LIN {X 0.108,Y -513.249,Z 696.655,A 0.000,B 0.000,C 90.000,E1 333.896} C_DIS
LIN {X -0.045,Y -530.728,Z 696.649,A 0.000,B 0.000,C 90.000,E1 332.743} C_DIS
LIN {X 0.068,Y -536.802,Z 696.646,A 0.000,B 0.000,C 90.000,E1 332.308} C_DIS
LIN {X -0.021,Y -544.293,Z 696.643,A 0.000,B 0.000,C 90.000,E1 331.769} C_DIS
LIN {X 0.058,Y -551.459,Z 696.640,A 0.000,B 0.000,C 90.000,E1 331.179} C_DIS
LIN {X -0.040,Y -558.208,Z 696.637,A 0.000,B 0.000,C 90.000,E1 330.589} C_DIS
LIN {X 0.004,Y -562.208,Z 696.635,A 0.000,B 0.000,C 90.000,E1 330.205} C_DIS
LIN {X -0.100,Y -567.315,Z 696.632,A 0.000,B 0.000,C 90.000,E1 329.715} C_DIS
LIN {X 0.042,Y -574.841,Z 696.627,A 0.000,B 0.000,C 90.000,E1 328.918} C_DIS
LIN {X -0.001,Y -583.472,Z 696.622,A 0.000,B 0.000,C 90.000,E1 327.995} C_DIS
LIN {X 0.085,Y -588.408,Z 696.619,A 0.000,B 0.000,C 90.000,E1 327.454} C_DIS
LIN {X 0.306,Y -596.576,Z 696.614,A 0.000,B 0.000,C 90.000,E1 326.501} C_DIS
LIN {X -0.095,Y -603.275,Z 696.610,A 0.000,B 0.000,C 90.000,E1 325.754} C_DIS
LIN {X -0.164,Y -609.504,Z 696.605,A 0.000,B 0.000,C 90.000,E1 324.975} C_DIS
LIN {X -0.135,Y -614.465,Z 696.602,A 0.000,B 0.000,C 90.000,E1 324.322} C_DIS
LIN {X -0.109,Y -620.766,Z 696.597,A 0.000,B 0.000,C 90.000,E1 323.417} C_DIS
LIN {X 0.004,Y -625.954,Z 696.592,A 0.000,B 0.000,C 90.000,E1 322.637} C_DIS
LIN {X 0.012,Y -633.084,Z 696.586,A 0.000,B 0.000,C 90.000,E1 321.492} C_DIS
LIN {X 0.145,Y -637.620,Z 696.582,A 0.000,B 0.000,C 90.000,E1 320.723} C_DIS
LIN {X -0.076,Y -641.917,Z 696.578,A 0.000,B 0.000,C 90.000,E1 319.989} C_DIS
LIN {X 0.082,Y -648.096,Z 696.571,A 0.000,B 0.000,C 90.000,E1 318.852} C_DIS
LIN {X -0.152,Y -653.942,Z 696.565,A 0.000,B 0.000,C 90.000,E1 317.757} C_DIS
LIN {X 0.212,Y -657.573,Z 696.561,A 0.000,B 0.000,C 90.000,E1 316.986} C_DIS
LIN {X -0.327,Y -660.960,Z 696.557,A 0.000,B 0.000,C 90.000,E1 316.296} C_DIS
LIN {X -0.383,Y -664.239,Z 696.553,A 0.000,B 0.000,C 90.000,E1 315.567} C_DIS
LIN {X 0.064,Y -668.154,Z 696.548,A 0.000,B 0.000,C 90.000,E1 314.555} C_DIS
LIN {X 0.123,Y -672.812,Z 696.541,A 0.000,B 0.000,C 90.000,E1 313.338} C_DIS
LIN {X 0.209,Y -676.430,Z 696.536,A 0.000,B 0.000,C 90.000,E1 312.366} C_DIS
LIN {X -0.126,Y -679.960,Z 696.530,A 0.000,B 0.000,C 90.000,E1 311.434} C_DIS
LIN {X 0.093,Y -683.151,Z 696.525,A 0.000,B 0.000,C 90.000,E1 310.458} C_DIS
LIN {X -0.079,Y -686.060,Z 696.520,A 0.000,B 0.000,C 90.000,E1 309.519} C_DIS
LIN {X 0.020,Y -687.452,Z 696.517,A 0.000,B 0.000,C 90.000,E1 309.036} C_DIS
LIN {X 0.279,Y -689.267,Z 696.513,A 0.000,B 0.000,C 90.000,E1 308.302} C_DIS
LIN {X 0.187,Y -691.415,Z 696.508,A 0.000,B 0.000,C 90.000,E1 307.363} C_DIS
LIN {X 0.068,Y -692.857,Z 696.504,A 0.000,B 0.000,C 90.000,E1 306.664} C_DIS
LIN {X -0.332,Y -695.101,Z 696.497,A 0.000,B 0.000,C 90.000,E1 305.518} C_DIS
LIN {X 0.160,Y -696.257,Z 696.493,A 0.000,B 0.000,C 90.000,E1 304.771} C_DIS
LIN {X 0.036,Y -698.131,Z 696.485,A 0.000,B 0.000,C 90.000,E1 303.372} C_DIS
LIN {X 0.229,Y -699.119,Z 696.480,A 0.000,B 0.000,C 90.000,E1 302.418} C_DIS
LIN {X -0.243,Y -700.440,Z 696.472,A 0.000,B 0.000,C 90.000,E1 301.052} C_DIS
LIN {X -0.053,Y -701.022,Z 696.469,A 0.000,B 0.000,C 90.000,E1 300.335} C_DIS
LIN {X -0.253,Y -701.671,Z 696.461,A 0.000,B 0.000,C 90.000,E1 298.949} C_DIS
LIN {X 0.101,Y -702.488,Z 696.450,A 0.000,B 0.000,C 90.000,E1 297.052} C_DIS
LIN {X -0.098,Y -703.278,Z 696.443,A 0.000,B 0.000,C 90.000,E1 295.668} C_DIS
LIN {X -0.168,Y -703.320,Z 696.440,A 0.000,B 0.000,C 90.000,E1 295.207} C_DIS
LIN {X 0.113,Y -703.122,Z 696.439,A 0.000,B 0.000,C 90.000,E1 294.951} C_DIS
LIN {X -0.259,Y -702.120,Z 696.436,A 0.000,B 0.000,C 90.000,E1 294.515} C_DIS
LIN {X 0.018,Y -701.136,Z 696.435,A 0.000,B 0.000,C 90.000,E1 294.259} C_DIS
LIN {X 0.007,Y -699.413,Z 696.434,A 0.000,B 0.000,C 90.000,E1 294.027} C_DIS
LIN {X 0.276,Y -697.550,Z 696.432,A 0.000,B 0.000,C 90.000,E1 293.770} C_DIS
LIN {X -0.231,Y -696.472,Z 696.432,A 0.000,B 0.000,C 90.000,E1 293.695} C_DIS
LIN {X -0.101,Y -694.838,Z 696.431,A 0.000,B 0.000,C 90.000,E1 293.567} C_DIS
LIN {X 0.346,Y -688.862,Z 696.429,A 0.000,B 0.000,C 90.000,E1 293.259} C_DIS
LIN {X 0.117,Y -686.900,Z 696.429,A 0.000,B 0.000,C 90.000,E1 293.206} C_DIS
LIN {X 0.010,Y -684.820,Z 696.429,A 0.000,B 0.000,C 90.000,E1 293.153} C_DIS
LIN {X -0.122,Y -678.094,Z 696.428,A 0.000,B 0.000,C 90.000,E1 293.025} C_DIS
LIN {X -0.139,Y -661.568,Z 696.427,A 0.000,B 0.000,C 90.000,E1 292.823} C_DIS
LIN {X 0.114,Y -647.822,Z 696.426,A 0.000,B 0.000,C 90.000,E1 292.589} C_DIS
LIN {X 0.091,Y -638.127,Z 696.425,A 0.000,B 0.000,C 90.000,E1 292.408} C_DIS
LIN {X 0.149,Y -624.755,Z 696.423,A 0.000,B 0.000,C 90.000,E1 292.099} C_DIS
LIN {X -0.052,Y -607.642,Z 696.420,A 0.000,B 0.000,C 90.000,E1 291.663} C_DIS
LIN {X -0.239,Y -576.587,Z 696.415,A 0.000,B 0.000,C 90.000,E1 290.737} C_DIS
LIN {X 0.266,Y -569.169,Z 696.414,A 0.000,B 0.000,C 90.000,E1 290.482} C_DIS
LIN {X 0.114,Y -563.221,Z 696.413,A 0.000,B 0.000,C 90.000,E1 290.301} C_DIS
LIN {X 0.212,Y -560.426,Z 696.412,A 0.000,B 0.000,C 90.000,E1 290.174} C_DIS
LIN {X 0.106,Y -558.042,Z 696.412,A 0.000,B 0.000,C 90.000,E1 290.066} C_DIS
LIN {X -0.099,Y -555.714,Z 696.410,A 0.000,B 0.000,C 90.000,E1 289.885} C_DIS
LIN {X -0.136,Y -555.678,Z 696.410,A 0.000,B 0.000,C 90.000,E1 289.885} C_DIS
LIN {X 0.246,Y -554.917,Z 696.409,A 0.000,B 0.000,C 90.000,E1 289.631} C_DIS
LIN {X 0.065,Y -554.334,Z 696.406,A 0.000,B 0.000,C 90.000,E1 289.087} C_DIS
LIN {X 0.062,Y -553.901,Z 696.398,A 0.000,B 0.000,C 90.000,E1 287.692} C_DIS
LIN {X -0.009,Y -553.252,Z 696.389,A 0.000,B 0.000,C 90.000,E1 286.024} C_DIS
LIN {X 0.070,Y -552.874,Z 696.383,A 0.000,B 0.000,C 90.000,E1 284.898} C_DIS
LIN {X -0.155,Y -552.256,Z 696.374,A 0.000,B 0.000,C 90.000,E1 283.244} C_DIS
LIN {X 0.018,Y -551.645,Z 696.366,A 0.000,B 0.000,C 90.000,E1 281.827} C_DIS
LIN {X 0.069,Y -550.859,Z 696.356,A 0.000,B 0.000,C 90.000,E1 280.141} C_DIS
LIN {X -0.298,Y -549.954,Z 696.344,A 0.000,B 0.000,C 90.000,E1 277.936} C_DIS
LIN {X -0.091,Y -549.215,Z 696.328,A 0.000,B 0.000,C 90.000,E1 275.106} C_DIS
LIN {X -0.203,Y -548.955,Z 696.317,A 0.000,B 0.000,C 90.000,E1 273.151} C_DIS
LIN {X -0.006,Y -548.668,Z 696.311,A 0.000,B 0.000,C 90.000,E1 272.007} C_DIS
LIN {X 0.160,Y -548.440,Z 696.307,A 0.000,B 0.000,C 90.000,E1 271.146} C_DIS
LIN {X -0.045,Y -547.378,Z 696.296,A 0.000,B 0.000,C 90.000,E1 269.198} C_DIS
LIN {X 0.235,Y -546.347,Z 696.286,A 0.000,B 0.000,C 90.000,E1 267.478} C_DIS
LIN {X -0.020,Y -545.246,Z 696.277,A 0.000,B 0.000,C 90.000,E1 265.812} C_DIS
LIN {X -0.227,Y -543.753,Z 696.266,A 0.000,B 0.000,C 90.000,E1 263.856} C_DIS
LIN {X -0.042,Y -542.813,Z 696.260,A 0.000,B 0.000,C 90.000,E1 262.704} C_DIS
LIN {X -0.193,Y -540.813,Z 696.248,A 0.000,B 0.000,C 90.000,E1 260.735} C_DIS
LIN {X -0.169,Y -538.511,Z 696.234,A 0.000,B 0.000,C 90.000,E1 258.173} C_DIS
LIN {X -0.123,Y -536.708,Z 696.223,A 0.000,B 0.000,C 90.000,E1 256.172} C_DIS
LIN {X 0.182,Y -536.028,Z 696.218,A 0.000,B 0.000,C 90.000,E1 255.283} C_DIS
LIN {X 0.249,Y -534.304,Z 696.209,A 0.000,B 0.000,C 90.000,E1 253.559} C_DIS
LIN {X -0.079,Y -532.474,Z 696.199,A 0.000,B 0.000,C 90.000,E1 251.873} C_DIS
LIN {X -0.152,Y -531.320,Z 696.193,A 0.000,B 0.000,C 90.000,E1 250.732} C_DIS
LIN {X -0.070,Y -530.084,Z 696.187,A 0.000,B 0.000,C 90.000,E1 249.571} C_DIS
LIN {X -0.133,Y -527.665,Z 696.177,A 0.000,B 0.000,C 90.000,E1 247.847} C_DIS
LIN {X 0.090,Y -525.999,Z 696.170,A 0.000,B 0.000,C 90.000,E1 246.666} C_DIS
LIN {X 0.119,Y -524.652,Z 696.166,A 0.000,B 0.000,C 90.000,E1 245.793} C_DIS
LIN {X -0.126,Y -521.764,Z 696.156,A 0.000,B 0.000,C 90.000,E1 244.076} C_DIS
LIN {X 0.218,Y -519.540,Z 696.149,A 0.000,B 0.000,C 90.000,E1 242.871} C_DIS
LIN {X -0.031,Y -516.692,Z 696.141,A 0.000,B 0.000,C 90.000,E1 241.435} C_DIS
LIN {X 0.016,Y -514.319,Z 696.135,A 0.000,B 0.000,C 90.000,E1 240.255} C_DIS
LIN {X -0.070,Y -511.228,Z 696.127,A 0.000,B 0.000,C 90.000,E1 238.791} C_DIS
LIN {X -0.219,Y -508.022,Z 696.118,A 0.000,B 0.000,C 90.000,E1 237.327} C_DIS
LIN {X 0.222,Y -505.390,Z 696.112,A 0.000,B 0.000,C 90.000,E1 236.087} C_DIS
LIN {X 0.096,Y -502.049,Z 696.104,A 0.000,B 0.000,C 90.000,E1 234.609} C_DIS
LIN {X 0.033,Y -499.257,Z 696.097,A 0.000,B 0.000,C 90.000,E1 233.417} C_DIS
LIN {X 0.223,Y -496.243,Z 696.090,A 0.000,B 0.000,C 90.000,E1 232.190} C_DIS
LIN {X 0.069,Y -490.251,Z 696.077,A 0.000,B 0.000,C 90.000,E1 229.784} C_DIS
LIN {X 0.022,Y -485.908,Z 696.066,A 0.000,B 0.000,C 90.000,E1 227.957} C_DIS
LIN {X -0.016,Y -481.004,Z 696.055,A 0.000,B 0.000,C 90.000,E1 225.810} C_DIS
LIN {X -0.189,Y -478.295,Z 696.048,A 0.000,B 0.000,C 90.000,E1 224.595} C_DIS
LIN {X 0.048,Y -474.759,Z 696.039,A 0.000,B 0.000,C 90.000,E1 223.014} C_DIS
LIN {X -0.103,Y -471.293,Z 696.030,A 0.000,B 0.000,C 90.000,E1 221.472} C_DIS
LIN {X 0.102,Y -467.176,Z 696.020,A 0.000,B 0.000,C 90.000,E1 219.564} C_DIS
LIN {X -0.020,Y -463.201,Z 696.009,A 0.000,B 0.000,C 90.000,E1 217.684} C_DIS
LIN {X -0.111,Y -458.072,Z 695.995,A 0.000,B 0.000,C 90.000,E1 215.152} C_DIS
LIN {X 0.306,Y -455.033,Z 695.986,A 0.000,B 0.000,C 90.000,E1 213.499} C_DIS
LIN {X 0.035,Y -451.969,Z 695.977,A 0.000,B 0.000,C 90.000,E1 211.926} C_DIS
LIN {X 0.012,Y -447.710,Z 695.965,A 0.000,B 0.000,C 90.000,E1 209.667} C_DIS
LIN {X 0.045,Y -443.555,Z 695.952,A 0.000,B 0.000,C 90.000,E1 207.385} C_DIS
LIN {X -0.122,Y -440.641,Z 695.943,A 0.000,B 0.000,C 90.000,E1 205.771} C_DIS
LIN {X -0.145,Y -437.670,Z 695.934,A 0.000,B 0.000,C 90.000,E1 204.131} C_DIS
LIN {X -0.168,Y -433.971,Z 695.923,A 0.000,B 0.000,C 90.000,E1 202.153} C_DIS
LIN {X -0.091,Y -430.969,Z 695.914,A 0.000,B 0.000,C 90.000,E1 200.482} C_DIS
LIN {X -0.028,Y -427.298,Z 695.903,A 0.000,B 0.000,C 90.000,E1 198.471} C_DIS
LIN {X -0.134,Y -423.137,Z 695.890,A 0.000,B 0.000,C 90.000,E1 196.134} C_DIS
LIN {X 0.011,Y -420.120,Z 695.880,A 0.000,B 0.000,C 90.000,E1 194.426} C_DIS
LIN {X -0.102,Y -415.938,Z 695.867,A 0.000,B 0.000,C 90.000,E1 192.063} C_DIS
LIN {X 0.217,Y -413.119,Z 695.857,A 0.000,B 0.000,C 90.000,E1 190.310} C_DIS
LIN {X 0.025,Y -409.762,Z 695.846,A 0.000,B 0.000,C 90.000,E1 188.276} C_DIS
LIN {X 0.049,Y -406.705,Z 695.835,A 0.000,B 0.000,C 90.000,E1 186.201} C_DIS
LIN {X -0.040,Y -403.260,Z 695.821,A 0.000,B 0.000,C 90.000,E1 183.784} C_DIS
LIN {X 0.025,Y -399.368,Z 695.804,A 0.000,B 0.000,C 90.000,E1 180.630} C_DIS
LIN {X -0.112,Y -395.946,Z 695.784,A 0.000,B 0.000,C 90.000,E1 177.135} C_DIS
LIN {X -0.171,Y -393.858,Z 695.768,A 0.000,B 0.000,C 90.000,E1 174.318} C_DIS
LIN {X 0.047,Y -392.119,Z 695.747,A 0.000,B 0.000,C 90.000,E1 170.387} C_DIS
LIN {X -0.203,Y -391.473,Z 695.733,A 0.000,B 0.000,C 90.000,E1 167.937} C_DIS
LIN {X 0.130,Y -390.914,Z 695.721,A 0.000,B 0.000,C 90.000,E1 165.755} C_DIS
LIN {X 0.146,Y -390.479,Z 695.705,A 0.000,B 0.000,C 90.000,E1 162.906} C_DIS
LIN {X -0.008,Y -390.447,Z 695.695,A 0.000,B 0.000,C 90.000,E1 161.148} C_DIS
LIN {X 0.061,Y -390.499,Z 695.681,A 0.000,B 0.000,C 90.000,E1 158.646} C_DIS
LIN {X -0.100,Y -390.667,Z 695.668,A 0.000,B 0.000,C 90.000,E1 156.177} C_DIS
LIN {X 0.213,Y -390.978,Z 695.654,A 0.000,B 0.000,C 90.000,E1 153.640} C_DIS
LIN {X 0.164,Y -391.240,Z 695.642,A 0.000,B 0.000,C 90.000,E1 151.513} C_DIS
LIN {X -0.185,Y -391.908,Z 695.628,A 0.000,B 0.000,C 90.000,E1 149.076} C_DIS
LIN {X 0.174,Y -392.559,Z 695.618,A 0.000,B 0.000,C 90.000,E1 147.248} C_DIS
LIN {X 0.153,Y -393.926,Z 695.604,A 0.000,B 0.000,C 90.000,E1 144.769} C_DIS
LIN {X 0.031,Y -394.813,Z 695.597,A 0.000,B 0.000,C 90.000,E1 143.371} C_DIS
LIN {X 0.035,Y -396.587,Z 695.585,A 0.000,B 0.000,C 90.000,E1 141.251} C_DIS
LIN {X 0.039,Y -398.612,Z 695.573,A 0.000,B 0.000,C 90.000,E1 139.138} C_DIS
LIN {X -0.021,Y -400.455,Z 695.563,A 0.000,B 0.000,C 90.000,E1 137.391} C_DIS
LIN {X -0.097,Y -401.201,Z 695.559,A 0.000,B 0.000,C 90.000,E1 136.701} C_DIS
LIN {X 0.108,Y -402.322,Z 695.556,A 0.000,B 0.000,C 90.000,E1 135.972} C_DIS
LIN {X -0.045,Y -404.292,Z 695.551,A 0.000,B 0.000,C 90.000,E1 135.121} C_DIS
LIN {X -0.117,Y -407.030,Z 695.547,A 0.000,B 0.000,C 90.000,E1 134.433} C_DIS
LIN {X 0.194,Y -409.182,Z 695.545,A 0.000,B 0.000,C 90.000,E1 134.028} C_DIS
LIN {X 0.022,Y -412.574,Z 695.542,A 0.000,B 0.000,C 90.000,E1 133.623} C_DIS
LIN {X -0.085,Y -418.142,Z 695.539,A 0.000,B 0.000,C 90.000,E1 133.056} C_DIS
LIN {X 0.040,Y -436.277,Z 695.530,A 0.000,B 0.000,C 90.000,E1 131.391} C_DIS
LIN {X -0.063,Y -454.811,Z 695.521,A 0.000,B 0.000,C 90.000,E1 129.850} C_DIS
LIN {X 0.035,Y -465.484,Z 695.516,A 0.000,B 0.000,C 90.000,E1 128.955} C_DIS
LIN {X 0.013,Y -474.374,Z 695.512,A 0.000,B 0.000,C 90.000,E1 128.177} C_DIS
LIN {X 0.078,Y -481.386,Z 695.509,A 0.000,B 0.000,C 90.000,E1 127.523} C_DIS
LIN {X -0.109,Y -488.508,Z 695.505,A 0.000,B 0.000,C 90.000,E1 126.870} C_DIS
LIN {X 0.152,Y -495.304,Z 695.501,A 0.000,B 0.000,C 90.000,E1 126.171} C_DIS
LIN {X 0.101,Y -502.112,Z 695.497,A 0.000,B 0.000,C 90.000,E1 125.471} C_DIS
LIN {X 0.044,Y -508.566,Z 695.493,A 0.000,B 0.000,C 90.000,E1 124.771} C_DIS
LIN {X 0.125,Y -513.389,Z 695.490,A 0.000,B 0.000,C 90.000,E1 124.199} C_DIS
LIN {X -0.011,Y -517.919,Z 695.487,A 0.000,B 0.000,C 90.000,E1 123.658} C_DIS
LIN {X 0.083,Y -522.141,Z 695.484,A 0.000,B 0.000,C 90.000,E1 123.086} C_DIS
LIN {X 0.009,Y -526.038,Z 695.481,A 0.000,B 0.000,C 90.000,E1 122.546} C_DIS
LIN {X -0.254,Y -530.643,Z 695.477,A 0.000,B 0.000,C 90.000,E1 121.878} C_DIS
LIN {X 0.146,Y -534.089,Z 695.474,A 0.000,B 0.000,C 90.000,E1 121.258} C_DIS
LIN {X 0.016,Y -538.708,Z 695.469,A 0.000,B 0.000,C 90.000,E1 120.413} C_DIS
LIN {X -0.128,Y -542.209,Z 695.465,A 0.000,B 0.000,C 90.000,E1 119.716} C_DIS
LIN {X -0.044,Y -545.486,Z 695.461,A 0.000,B 0.000,C 90.000,E1 118.999} C_DIS
LIN {X 0.071,Y -548.557,Z 695.457,A 0.000,B 0.000,C 90.000,E1 118.281} C_DIS
LIN {X -0.161,Y -551.986,Z 695.453,A 0.000,B 0.000,C 90.000,E1 117.462} C_DIS
LIN {X -0.102,Y -555.184,Z 695.448,A 0.000,B 0.000,C 90.000,E1 116.616} C_DIS
LIN {X 0.277,Y -559.133,Z 695.442,A 0.000,B 0.000,C 90.000,E1 115.463} C_DIS
LIN {X 0.164,Y -561.826,Z 695.437,A 0.000,B 0.000,C 90.000,E1 114.643} C_DIS
LIN {X 0.080,Y -564.293,Z 695.432,A 0.000,B 0.000,C 90.000,E1 113.823} C_DIS
LIN {X 0.128,Y -567.059,Z 695.426,A 0.000,B 0.000,C 90.000,E1 112.717} C_DIS
LIN {X -0.247,Y -568.297,Z 695.423,A 0.000,B 0.000,C 90.000,E1 112.206} C_DIS
LIN {X -0.139,Y -570.468,Z 695.417,A 0.000,B 0.000,C 90.000,E1 111.099} C_DIS
LIN {X 0.162,Y -572.974,Z 695.410,A 0.000,B 0.000,C 90.000,E1 109.704} C_DIS
LIN {X -0.032,Y -575.321,Z 695.402,A 0.000,B 0.000,C 90.000,E1 108.362} C_DIS
LIN {X 0.180,Y -577.652,Z 695.395,A 0.000,B 0.000,C 90.000,E1 106.985} C_DIS
LIN {X 0.222,Y -579.456,Z 695.388,A 0.000,B 0.000,C 90.000,E1 105.898} C_DIS
LIN {X -0.218,Y -581.581,Z 695.381,A 0.000,B 0.000,C 90.000,E1 104.592} C_DIS
LIN {X 0.173,Y -584.094,Z 695.372,A 0.000,B 0.000,C 90.000,E1 102.939} C_DIS
LIN {X -0.205,Y -586.524,Z 695.363,A 0.000,B 0.000,C 90.000,E1 101.366} C_DIS
LIN {X -0.096,Y -588.661,Z 695.356,A 0.000,B 0.000,C 90.000,E1 100.018} C_DIS
LIN {X 0.258,Y -590.190,Z 695.350,A 0.000,B 0.000,C 90.000,E1 98.916} C_DIS
LIN {X 0.049,Y -591.654,Z 695.344,A 0.000,B 0.000,C 90.000,E1 97.871} C_DIS
LIN {X 0.241,Y -593.679,Z 695.335,A 0.000,B 0.000,C 90.000,E1 96.258} C_DIS
LIN {X 0.213,Y -595.276,Z 695.328,A 0.000,B 0.000,C 90.000,E1 94.935} C_DIS
LIN {X 0.211,Y -596.785,Z 695.320,A 0.000,B 0.000,C 90.000,E1 93.612} C_DIS
LIN {X -0.036,Y -597.871,Z 695.314,A 0.000,B 0.000,C 90.000,E1 92.579} C_DIS
LIN {X -0.274,Y -598.771,Z 695.308,A 0.000,B 0.000,C 90.000,E1 91.547} C_DIS
LIN {X 0.083,Y -599.562,Z 695.303,A 0.000,B 0.000,C 90.000,E1 90.458} C_DIS
LIN {X 0.098,Y -600.276,Z 695.295,A 0.000,B 0.000,C 90.000,E1 89.141} C_DIS
LIN {X 0.138,Y -600.768,Z 695.288,A 0.000,B 0.000,C 90.000,E1 87.822} C_DIS
LIN {X -0.055,Y -601.030,Z 695.282,A 0.000,B 0.000,C 90.000,E1 86.788} C_DIS
LIN {X -0.003,Y -601.236,Z 695.275,A 0.000,B 0.000,C 90.000,E1 85.469} C_DIS
LIN {X -0.146,Y -601.240,Z 695.269,A 0.000,B 0.000,C 90.000,E1 84.432} C_DIS
LIN {X 0.315,Y -601.145,Z 695.263,A 0.000,B 0.000,C 90.000,E1 83.337} C_DIS
LIN {X 0.174,Y -600.969,Z 695.257,A 0.000,B 0.000,C 90.000,E1 82.299} C_DIS
LIN {X 0.111,Y -600.661,Z 695.252,A 0.000,B 0.000,C 90.000,E1 81.254} C_DIS
LIN {X 0.049,Y -600.044,Z 695.246,A 0.000,B 0.000,C 90.000,E1 80.208} C_DIS
LIN {X -0.023,Y -599.215,Z 695.240,A 0.000,B 0.000,C 90.000,E1 79.162} C_DIS
LIN {X 0.178,Y -598.089,Z 695.232,A 0.000,B 0.000,C 90.000,E1 77.825} C_DIS
LIN {X 0.185,Y -597.114,Z 695.227,A 0.000,B 0.000,C 90.000,E1 76.769} C_DIS
LIN {X -0.268,Y -595.454,Z 695.218,A 0.000,B 0.000,C 90.000,E1 75.227} C_DIS
LIN {X 0.123,Y -593.924,Z 695.211,A 0.000,B 0.000,C 90.000,E1 73.866} C_DIS
LIN {X 0.082,Y -592.318,Z 695.203,A 0.000,B 0.000,C 90.000,E1 72.543} C_DIS
LIN {X 0.013,Y -590.482,Z 695.196,A 0.000,B 0.000,C 90.000,E1 71.221} C_DIS
LIN {X -0.021,Y -588.015,Z 695.187,A 0.000,B 0.000,C 90.000,E1 69.625} C_DIS
LIN {X 0.156,Y -586.212,Z 695.181,A 0.000,B 0.000,C 90.000,E1 68.539} C_DIS
LIN {X -0.032,Y -584.174,Z 695.175,A 0.000,B 0.000,C 90.000,E1 67.486} C_DIS
LIN {X -0.015,Y -581.818,Z 695.169,A 0.000,B 0.000,C 90.000,E1 66.410} C_DIS
LIN {X -0.262,Y -579.215,Z 695.163,A 0.000,B 0.000,C 90.000,E1 65.357} C_DIS
LIN {X -0.161,Y -577.083,Z 695.159,A 0.000,B 0.000,C 90.000,E1 64.537} C_DIS
LIN {X -0.088,Y -574.755,Z 695.154,A 0.000,B 0.000,C 90.000,E1 63.717} C_DIS
LIN {X 0.216,Y -572.228,Z 695.149,A 0.000,B 0.000,C 90.000,E1 62.871} C_DIS
LIN {X 0.325,Y -568.637,Z 695.143,A 0.000,B 0.000,C 90.000,E1 61.769} C_DIS
LIN {X 0.069,Y -565.689,Z 695.139,A 0.000,B 0.000,C 90.000,E1 60.973} C_DIS
LIN {X 0.277,Y -562.505,Z 695.134,A 0.000,B 0.000,C 90.000,E1 60.127} C_DIS
LIN {X -0.037,Y -558.888,Z 695.130,A 0.000,B 0.000,C 90.000,E1 59.331} C_DIS
LIN {X 0.190,Y -555.551,Z 695.126,A 0.000,B 0.000,C 90.000,E1 58.614} C_DIS
LIN {X 0.027,Y -552.644,Z 695.123,A 0.000,B 0.000,C 90.000,E1 58.074} C_DIS
LIN {X 0.018,Y -548.514,Z 695.119,A 0.000,B 0.000,C 90.000,E1 57.375} C_DIS
LIN {X -0.321,Y -544.014,Z 695.115,A 0.000,B 0.000,C 90.000,E1 56.707} C_DIS
LIN {X 0.189,Y -540.056,Z 695.112,A 0.000,B 0.000,C 90.000,E1 56.087} C_DIS
LIN {X -0.082,Y -535.707,Z 695.109,A 0.000,B 0.000,C 90.000,E1 55.548} C_DIS
LIN {X 0.103,Y -532.117,Z 695.106,A 0.000,B 0.000,C 90.000,E1 55.102} C_DIS
LIN {X -0.213,Y -527.228,Z 695.103,A 0.000,B 0.000,C 90.000,E1 54.609} C_DIS
LIN {X 0.155,Y -522.068,Z 695.101,A 0.000,B 0.000,C 90.000,E1 54.069} C_DIS
LIN {X -0.166,Y -516.546,Z 695.098,A 0.000,B 0.000,C 90.000,E1 53.623} C_DIS
LIN {X 0.201,Y -511.623,Z 695.096,A 0.000,B 0.000,C 90.000,E1 53.210} C_DIS
LIN {X 0.236,Y -505.365,Z 695.093,A 0.000,B 0.000,C 90.000,E1 52.763} C_DIS
LIN {X -0.126,Y -498.968,Z 695.091,A 0.000,B 0.000,C 90.000,E1 52.396} C_DIS
LIN {X 0.068,Y -489.097,Z 695.088,A 0.000,B 0.000,C 90.000,E1 51.778} C_DIS
LIN {X -0.109,Y -474.324,Z 695.083,A 0.000,B 0.000,C 90.000,E1 50.964} C_DIS
LIN {X -0.007,Y -467.665,Z 695.081,A 0.000,B 0.000,C 90.000,E1 50.561} C_DIS
LIN {X -0.061,Y -457.921,Z 695.078,A 0.000,B 0.000,C 90.000,E1 49.989} C_DIS
LIN {X -0.011,Y -440.182,Z 695.072,A 0.000,B 0.000,C 90.000,E1 48.895} C_DIS
LIN {X 0.011,Y -431.973,Z 695.069,A 0.000,B 0.000,C 90.000,E1 48.366} C_DIS
LIN {X 0.061,Y -424.375,Z 695.066,A 0.000,B 0.000,C 90.000,E1 47.796} C_DIS
LIN {X 0.033,Y -424.361,Z 695.066,A 0.000,B 0.000,C 90.000,E1 47.796} C_DIS
LIN {X 0.137,Y -418.983,Z 695.050,A 0.000,B 0.000,C 90.000,E1 45.000} C_DIS
LIN {X 0.026,Y -418.304,Z 695.048,A 0.000,B 0.000,C 90.000,E1 44.676} C_DIS
LIN {X 0.079,Y -411.430,Z 695.031,A 0.000,B 0.000,C 90.000,E1 41.595} C_DIS
LIN {X -0.158,Y -411.330,Z 695.024,A 0.000,B 0.000,C 90.000,E1 40.253} C_DIS
LIN {X 0.019,Y -411.919,Z 695.004,A 0.000,B 0.000,C 90.000,E1 36.790} C_DIS
LIN {X -0.053,Y -412.776,Z 694.993,A 0.000,B 0.000,C 90.000,E1 34.739} C_DIS
LIN {X -0.001,Y -413.750,Z 694.982,A 0.000,B 0.000,C 90.000,E1 32.673} C_DIS
LIN {X 0.261,Y -414.647,Z 694.972,A 0.000,B 0.000,C 90.000,E1 30.924} C_DIS
LIN {X -0.235,Y -415.608,Z 694.963,A 0.000,B 0.000,C 90.000,E1 29.283} C_DIS
LIN {X -0.084,Y -417.030,Z 694.949,A 0.000,B 0.000,C 90.000,E1 26.873} C_DIS
LIN {X 0.104,Y -418.712,Z 694.936,A 0.000,B 0.000,C 90.000,E1 24.463} C_DIS
LIN {X 0.107,Y -421.365,Z 694.919,A 0.000,B 0.000,C 90.000,E1 21.408} C_DIS
LIN {X -0.199,Y -423.013,Z 694.910,A 0.000,B 0.000,C 90.000,E1 19.758} C_DIS
LIN {X -0.077,Y -424.691,Z 694.900,A 0.000,B 0.000,C 90.000,E1 18.055} C_DIS
LIN {X 0.013,Y -426.775,Z 694.889,A 0.000,B 0.000,C 90.000,E1 16.024} C_DIS
LIN {X 0.244,Y -429.414,Z 694.876,A 0.000,B 0.000,C 90.000,E1 13.647} C_DIS
LIN {X 0.027,Y -431.453,Z 694.867,A 0.000,B 0.000,C 90.000,E1 12.007} C_DIS
LIN {X 0.093,Y -434.331,Z 694.854,A 0.000,B 0.000,C 90.000,E1 9.670} C_DIS
LIN {X -0.125,Y -438.203,Z 694.837,A 0.000,B 0.000,C 90.000,E1 6.720} C_DIS
LIN {X -0.012,Y -441.878,Z 694.823,A 0.000,B 0.000,C 90.000,E1 4.073} C_DIS
LIN {X -0.127,Y -446.523,Z 694.806,A 0.000,B 0.000,C 90.000,E1 1.146} C_DIS
LIN {X 0.061,Y -451.737,Z 694.790,A 0.000,B 0.000,C 90.000,E1 358.165} C_DIS
LIN {X 0.181,Y -455.413,Z 694.779,A 0.000,B 0.000,C 90.000,E1 356.216} C_DIS
LIN {X -0.236,Y -458.539,Z 694.770,A 0.000,B 0.000,C 90.000,E1 354.666} C_DIS
LIN {X 0.177,Y -461.137,Z 694.763,A 0.000,B 0.000,C 90.000,E1 353.337} C_DIS
LIN {X 0.164,Y -464.841,Z 694.753,A 0.000,B 0.000,C 90.000,E1 351.432} C_DIS
LIN {X 0.104,Y -467.813,Z 694.744,A 0.000,B 0.000,C 90.000,E1 349.859} C_DIS
LIN {X 0.106,Y -470.644,Z 694.735,A 0.000,B 0.000,C 90.000,E1 348.285} C_DIS
LIN {X 0.255,Y -473.485,Z 694.726,A 0.000,B 0.000,C 90.000,E1 346.700} C_DIS
LIN {X -0.051,Y -476.955,Z 694.716,A 0.000,B 0.000,C 90.000,E1 344.866} C_DIS
LIN {X 0.150,Y -481.136,Z 694.704,A 0.000,B 0.000,C 90.000,E1 342.670} C_DIS
LIN {X -0.029,Y -484.162,Z 694.695,A 0.000,B 0.000,C 90.000,E1 341.148} C_DIS
LIN {X -0.140,Y -487.297,Z 694.687,A 0.000,B 0.000,C 90.000,E1 339.625} C_DIS
LIN {X -0.171,Y -491.077,Z 694.677,A 0.000,B 0.000,C 90.000,E1 337.794} C_DIS
LIN {X 0.164,Y -493.752,Z 694.670,A 0.000,B 0.000,C 90.000,E1 336.538} C_DIS
LIN {X 0.252,Y -495.390,Z 694.666,A 0.000,B 0.000,C 90.000,E1 335.921} C_DIS
LIN {X -0.090,Y -497.607,Z 694.663,A 0.000,B 0.000,C 90.000,E1 335.357} C_DIS
LIN {X 0.009,Y -499.063,Z 694.661,A 0.000,B 0.000,C 90.000,E1 335.049} C_DIS
LIN {X 0.055,Y -501.270,Z 694.660,A 0.000,B 0.000,C 90.000,E1 334.717} C_DIS
LIN {X 0.074,Y -505.386,Z 694.657,A 0.000,B 0.000,C 90.000,E1 334.280} C_DIS
LIN {X 0.145,Y -510.759,Z 694.655,A 0.000,B 0.000,C 90.000,E1 333.845} C_DIS
LIN {X 0.160,Y -517.047,Z 694.652,A 0.000,B 0.000,C 90.000,E1 333.384} C_DIS
LIN {X 0.019,Y -529.596,Z 694.648,A 0.000,B 0.000,C 90.000,E1 332.564} C_DIS
LIN {X 0.140,Y -537.285,Z 694.645,A 0.000,B 0.000,C 90.000,E1 332.025} C_DIS
LIN {X -0.213,Y -544.685,Z 694.642,A 0.000,B 0.000,C 90.000,E1 331.513} C_DIS
LIN {X -0.189,Y -550.344,Z 694.639,A 0.000,B 0.000,C 90.000,E1 331.051} C_DIS
LIN {X 0.119,Y -557.227,Z 694.636,A 0.000,B 0.000,C 90.000,E1 330.411} C_DIS
LIN {X -0.002,Y -563.949,Z 694.632,A 0.000,B 0.000,C 90.000,E1 329.793} C_DIS
LIN {X 0.083,Y -572.921,Z 694.627,A 0.000,B 0.000,C 90.000,E1 328.869} C_DIS
LIN {X 0.012,Y -581.672,Z 694.622,A 0.000,B 0.000,C 90.000,E1 327.946} C_DIS
LIN {X -0.115,Y -587.830,Z 694.618,A 0.000,B 0.000,C 90.000,E1 327.296} C_DIS
LIN {X 0.117,Y -596.054,Z 694.613,A 0.000,B 0.000,C 90.000,E1 326.342} C_DIS
LIN {X -0.063,Y -604.011,Z 694.608,A 0.000,B 0.000,C 90.000,E1 325.435} C_DIS
LIN {X -0.154,Y -611.229,Z 694.603,A 0.000,B 0.000,C 90.000,E1 324.529} C_DIS
LIN {X 0.064,Y -615.046,Z 694.600,A 0.000,B 0.000,C 90.000,E1 323.989} C_DIS
LIN {X 0.254,Y -620.453,Z 694.596,A 0.000,B 0.000,C 90.000,E1 323.210} C_DIS
LIN {X -0.110,Y -624.824,Z 694.592,A 0.000,B 0.000,C 90.000,E1 322.603} C_DIS
LIN {X 0.401,Y -631.292,Z 694.587,A 0.000,B 0.000,C 90.000,E1 321.537} C_DIS
LIN {X -0.252,Y -634.418,Z 694.584,A 0.000,B 0.000,C 90.000,E1 321.090} C_DIS
LIN {X -0.108,Y -639.621,Z 694.579,A 0.000,B 0.000,C 90.000,E1 320.194} C_DIS
LIN {X 0.020,Y -645.916,Z 694.573,A 0.000,B 0.000,C 90.000,E1 319.057} C_DIS
LIN {X -0.123,Y -649.291,Z 694.569,A 0.000,B 0.000,C 90.000,E1 318.447} C_DIS
LIN {X -0.294,Y -654.457,Z 694.564,A 0.000,B 0.000,C 90.000,E1 317.472} C_DIS
LIN {X 0.103,Y -656.901,Z 694.561,A 0.000,B 0.000,C 90.000,E1 316.944} C_DIS
LIN {X 0.009,Y -660.345,Z 694.557,A 0.000,B 0.000,C 90.000,E1 316.215} C_DIS
LIN {X -0.051,Y -663.645,Z 694.553,A 0.000,B 0.000,C 90.000,E1 315.486} C_DIS
LIN {X -0.078,Y -667.626,Z 694.547,A 0.000,B 0.000,C 90.000,E1 314.514} C_DIS
LIN {X -0.057,Y -671.427,Z 694.542,A 0.000,B 0.000,C 90.000,E1 313.542} C_DIS
LIN {X 0.068,Y -676.057,Z 694.535,A 0.000,B 0.000,C 90.000,E1 312.324} C_DIS
LIN {X -0.265,Y -679.597,Z 694.530,A 0.000,B 0.000,C 90.000,E1 311.391} C_DIS
LIN {X 0.359,Y -682.106,Z 694.526,A 0.000,B 0.000,C 90.000,E1 310.620} C_DIS
LIN {X -0.350,Y -685.122,Z 694.521,A 0.000,B 0.000,C 90.000,E1 309.725} C_DIS
LIN {X -0.111,Y -687.253,Z 694.517,A 0.000,B 0.000,C 90.000,E1 308.991} C_DIS
LIN {X 0.203,Y -689.622,Z 694.511,A 0.000,B 0.000,C 90.000,E1 308.016} C_DIS
LIN {X 0.064,Y -691.278,Z 694.507,A 0.000,B 0.000,C 90.000,E1 307.317} C_DIS
LIN {X 0.362,Y -692.734,Z 694.503,A 0.000,B 0.000,C 90.000,E1 306.583} C_DIS
LIN {X -0.042,Y -695.026,Z 694.497,A 0.000,B 0.000,C 90.000,E1 305.438} C_DIS
LIN {X -0.125,Y -696.218,Z 694.493,A 0.000,B 0.000,C 90.000,E1 304.739} C_DIS
LIN {X 0.319,Y -698.112,Z 694.485,A 0.000,B 0.000,C 90.000,E1 303.293} C_DIS
LIN {X -0.117,Y -698.897,Z 694.481,A 0.000,B 0.000,C 90.000,E1 302.625} C_DIS
LIN {X -0.330,Y -700.497,Z 694.472,A 0.000,B 0.000,C 90.000,E1 301.003} C_DIS
LIN {X 0.219,Y -701.054,Z 694.468,A 0.000,B 0.000,C 90.000,E1 300.256} C_DIS
LIN {X 0.014,Y -701.741,Z 694.460,A 0.000,B 0.000,C 90.000,E1 298.871} C_DIS
LIN {X 0.042,Y -702.598,Z 694.450,A 0.000,B 0.000,C 90.000,E1 297.001} C_DIS
LIN {X -0.125,Y -703.305,Z 694.444,A 0.000,B 0.000,C 90.000,E1 295.848} C_DIS
LIN {X 0.439,Y -703.430,Z 694.441,A 0.000,B 0.000,C 90.000,E1 295.335} C_DIS
LIN {X -0.214,Y -703.397,Z 694.440,A 0.000,B 0.000,C 90.000,E1 295.155} C_DIS
LIN {X 0.069,Y -703.044,Z 694.438,A 0.000,B 0.000,C 90.000,E1 294.899} C_DIS
LIN {X -0.300,Y -701.959,Z 694.436,A 0.000,B 0.000,C 90.000,E1 294.463} C_DIS
LIN {X -0.161,Y -701.477,Z 694.435,A 0.000,B 0.000,C 90.000,E1 294.335} C_DIS
LIN {X -0.023,Y -700.713,Z 694.435,A 0.000,B 0.000,C 90.000,E1 294.207} C_DIS
LIN {X -0.404,Y -696.897,Z 694.432,A 0.000,B 0.000,C 90.000,E1 293.770} C_DIS
LIN {X -0.273,Y -695.571,Z 694.431,A 0.000,B 0.000,C 90.000,E1 293.643} C_DIS
LIN {X -0.144,Y -693.432,Z 694.431,A 0.000,B 0.000,C 90.000,E1 293.515} C_DIS
LIN {X 0.053,Y -687.820,Z 694.429,A 0.000,B 0.000,C 90.000,E1 293.259} C_DIS
LIN {X -0.166,Y -685.468,Z 694.429,A 0.000,B 0.000,C 90.000,E1 293.206} C_DIS
LIN {X -0.322,Y -678.893,Z 694.428,A 0.000,B 0.000,C 90.000,E1 293.078} C_DIS
LIN {X 0.077,Y -661.290,Z 694.427,A 0.000,B 0.000,C 90.000,E1 292.823} C_DIS
LIN {X -0.284,Y -647.520,Z 694.426,A 0.000,B 0.000,C 90.000,E1 292.642} C_DIS
LIN {X -0.320,Y -637.894,Z 694.425,A 0.000,B 0.000,C 90.000,E1 292.461} C_DIS
LIN {X -0.294,Y -624.415,Z 694.423,A 0.000,B 0.000,C 90.000,E1 292.153} C_DIS
LIN {X 0.071,Y -607.299,Z 694.420,A 0.000,B 0.000,C 90.000,E1 291.663} C_DIS
LIN {X -0.186,Y -576.094,Z 694.415,A 0.000,B 0.000,C 90.000,E1 290.737} C_DIS
LIN {X 0.291,Y -568.636,Z 694.414,A 0.000,B 0.000,C 90.000,E1 290.482} C_DIS
LIN {X 0.125,Y -562.420,Z 694.413,A 0.000,B 0.000,C 90.000,E1 290.301} C_DIS
LIN {X -0.240,Y -557.929,Z 694.412,A 0.000,B 0.000,C 90.000,E1 290.120} C_DIS
LIN {X 0.110,Y -555.662,Z 694.411,A 0.000,B 0.000,C 90.000,E1 289.885} C_DIS
LIN {X 0.073,Y -555.636,Z 694.411,A 0.000,B 0.000,C 90.000,E1 289.885} C_DIS
LIN {X 0.271,Y -554.841,Z 694.409,A 0.000,B 0.000,C 90.000,E1 289.631} C_DIS
LIN {X -0.269,Y -554.389,Z 694.407,A 0.000,B 0.000,C 90.000,E1 289.268} C_DIS
LIN {X 0.256,Y -553.944,Z 694.399,A 0.000,B 0.000,C 90.000,E1 287.819} C_DIS
LIN {X -0.073,Y -553.195,Z 694.388,A 0.000,B 0.000,C 90.000,E1 285.898} C_DIS
LIN {X -0.116,Y -552.927,Z 694.384,A 0.000,B 0.000,C 90.000,E1 285.064} C_DIS
LIN {X 0.186,Y -552.293,Z 694.374,A 0.000,B 0.000,C 90.000,E1 283.355} C_DIS
LIN {X 0.239,Y -551.691,Z 694.367,A 0.000,B 0.000,C 90.000,E1 281.951} C_DIS
LIN {X -0.031,Y -550.765,Z 694.356,A 0.000,B 0.000,C 90.000,E1 280.018} C_DIS
LIN {X 0.131,Y -549.867,Z 694.343,A 0.000,B 0.000,C 90.000,E1 277.757} C_DIS
LIN {X 0.226,Y -549.232,Z 694.329,A 0.000,B 0.000,C 90.000,E1 275.220} C_DIS
LIN {X 0.081,Y -548.990,Z 694.318,A 0.000,B 0.000,C 90.000,E1 273.269} C_DIS
LIN {X -0.241,Y -548.751,Z 694.312,A 0.000,B 0.000,C 90.000,E1 272.178} C_DIS
LIN {X -0.023,Y -548.395,Z 694.306,A 0.000,B 0.000,C 90.000,E1 271.031} C_DIS
LIN {X 0.271,Y -547.488,Z 694.296,A 0.000,B 0.000,C 90.000,E1 269.312} C_DIS
LIN {X 0.010,Y -546.474,Z 694.287,A 0.000,B 0.000,C 90.000,E1 267.650} C_DIS
LIN {X -0.279,Y -545.392,Z 694.278,A 0.000,B 0.000,C 90.000,E1 265.988} C_DIS
LIN {X 0.002,Y -544.292,Z 694.270,A 0.000,B 0.000,C 90.000,E1 264.546} C_DIS
LIN {X 0.200,Y -543.482,Z 694.263,A 0.000,B 0.000,C 90.000,E1 263.394} C_DIS
LIN {X -0.159,Y -542.381,Z 694.257,A 0.000,B 0.000,C 90.000,E1 262.299} C_DIS
LIN {X 0.137,Y -540.662,Z 694.248,A 0.000,B 0.000,C 90.000,E1 260.566} C_DIS
LIN {X 0.254,Y -538.412,Z 694.234,A 0.000,B 0.000,C 90.000,E1 257.993} C_DIS
LIN {X 0.302,Y -536.615,Z 694.222,A 0.000,B 0.000,C 90.000,E1 255.992} C_DIS
LIN {X -0.049,Y -535.893,Z 694.218,A 0.000,B 0.000,C 90.000,E1 255.172} C_DIS
LIN {X -0.034,Y -534.476,Z 694.210,A 0.000,B 0.000,C 90.000,E1 253.740} C_DIS
LIN {X 0.148,Y -532.653,Z 694.200,A 0.000,B 0.000,C 90.000,E1 252.000} C_DIS
LIN {X 0.266,Y -531.195,Z 694.192,A 0.000,B 0.000,C 90.000,E1 250.550} C_DIS
LIN {X -0.151,Y -529.926,Z 694.186,A 0.000,B 0.000,C 90.000,E1 249.444} C_DIS
LIN {X -0.036,Y -527.113,Z 694.175,A 0.000,B 0.000,C 90.000,E1 247.411} C_DIS
LIN {X 0.179,Y -525.411,Z 694.168,A 0.000,B 0.000,C 90.000,E1 246.230} C_DIS
LIN {X -0.273,Y -522.510,Z 694.158,A 0.000,B 0.000,C 90.000,E1 244.537} C_DIS
LIN {X -0.064,Y -520.978,Z 694.154,A 0.000,B 0.000,C 90.000,E1 243.640} C_DIS
LIN {X 0.172,Y -518.145,Z 694.145,A 0.000,B 0.000,C 90.000,E1 242.153} C_DIS
LIN {X -0.100,Y -515.285,Z 694.137,A 0.000,B 0.000,C 90.000,E1 240.717} C_DIS
LIN {X 0.273,Y -512.170,Z 694.129,A 0.000,B 0.000,C 90.000,E1 239.203} C_DIS
LIN {X 0.138,Y -509.033,Z 694.121,A 0.000,B 0.000,C 90.000,E1 237.740} C_DIS
LIN {X -0.110,Y -506.401,Z 694.114,A 0.000,B 0.000,C 90.000,E1 236.580} C_DIS
LIN {X -0.221,Y -503.070,Z 694.106,A 0.000,B 0.000,C 90.000,E1 235.102} C_DIS
LIN {X -0.265,Y -500.283,Z 694.099,A 0.000,B 0.000,C 90.000,E1 233.909} C_DIS
LIN {X 0.070,Y -498.126,Z 694.094,A 0.000,B 0.000,C 90.000,E1 232.970} C_DIS
LIN {X -0.061,Y -495.077,Z 694.088,A 0.000,B 0.000,C 90.000,E1 231.778} C_DIS
LIN {X -0.315,Y -490.630,Z 694.078,A 0.000,B 0.000,C 90.000,E1 229.989} C_DIS
LIN {X 0.019,Y -486.287,Z 694.067,A 0.000,B 0.000,C 90.000,E1 228.119} C_DIS
LIN {X -0.146,Y -482.021,Z 694.057,A 0.000,B 0.000,C 90.000,E1 226.296} C_DIS
LIN {X -0.181,Y -478.626,Z 694.049,A 0.000,B 0.000,C 90.000,E1 224.757} C_DIS
LIN {X 0.063,Y -475.069,Z 694.040,A 0.000,B 0.000,C 90.000,E1 223.176} C_DIS
LIN {X 0.090,Y -470.203,Z 694.028,A 0.000,B 0.000,C 90.000,E1 220.987} C_DIS
LIN {X -0.039,Y -466.112,Z 694.017,A 0.000,B 0.000,C 90.000,E1 219.116} C_DIS
LIN {X 0.061,Y -462.803,Z 694.009,A 0.000,B 0.000,C 90.000,E1 217.523} C_DIS
LIN {X 0.061,Y -457.733,Z 693.994,A 0.000,B 0.000,C 90.000,E1 214.978} C_DIS
LIN {X -0.001,Y -455.338,Z 693.987,A 0.000,B 0.000,C 90.000,E1 213.706} C_DIS
LIN {X -0.172,Y -451.644,Z 693.977,A 0.000,B 0.000,C 90.000,E1 211.799} C_DIS
LIN {X -0.275,Y -447.987,Z 693.966,A 0.000,B 0.000,C 90.000,E1 209.873} C_DIS
LIN {X -0.020,Y -443.819,Z 693.953,A 0.000,B 0.000,C 90.000,E1 207.564} C_DIS
LIN {X 0.017,Y -440.908,Z 693.944,A 0.000,B 0.000,C 90.000,E1 205.924} C_DIS
LIN {X 0.029,Y -437.325,Z 693.933,A 0.000,B 0.000,C 90.000,E1 203.951} C_DIS
LIN {X -0.230,Y -434.259,Z 693.924,A 0.000,B 0.000,C 90.000,E1 202.333} C_DIS
LIN {X 0.071,Y -430.660,Z 693.913,A 0.000,B 0.000,C 90.000,E1 200.301} C_DIS
LIN {X -0.008,Y -426.949,Z 693.902,A 0.000,B 0.000,C 90.000,E1 198.308} C_DIS
LIN {X -0.108,Y -422.812,Z 693.889,A 0.000,B 0.000,C 90.000,E1 195.969} C_DIS
LIN {X 0.145,Y -419.825,Z 693.879,A 0.000,B 0.000,C 90.000,E1 194.245} C_DIS
LIN {X 0.017,Y -415.660,Z 693.866,A 0.000,B 0.000,C 90.000,E1 191.883} C_DIS
LIN {X -0.155,Y -412.855,Z 693.857,A 0.000,B 0.000,C 90.000,E1 190.197} C_DIS
LIN {X 0.061,Y -409.558,Z 693.845,A 0.000,B 0.000,C 90.000,E1 188.106} C_DIS
LIN {X 0.084,Y -406.485,Z 693.834,A 0.000,B 0.000,C 90.000,E1 186.030} C_DIS
LIN {X 0.030,Y -403.544,Z 693.822,A 0.000,B 0.000,C 90.000,E1 183.955} C_DIS
LIN {X 0.103,Y -399.632,Z 693.805,A 0.000,B 0.000,C 90.000,E1 180.802} C_DIS
LIN {X 0.038,Y -396.479,Z 693.787,A 0.000,B 0.000,C 90.000,E1 177.650} C_DIS
LIN {X -0.031,Y -394.315,Z 693.771,A 0.000,B 0.000,C 90.000,E1 174.837} C_DIS
LIN {X 0.102,Y -392.308,Z 693.748,A 0.000,B 0.000,C 90.000,E1 170.566} C_DIS
LIN {X -0.069,Y -391.672,Z 693.734,A 0.000,B 0.000,C 90.000,E1 168.105} C_DIS
LIN {X 0.145,Y -391.246,Z 693.724,A 0.000,B 0.000,C 90.000,E1 166.297} C_DIS
LIN {X -0.170,Y -390.713,Z 693.706,A 0.000,B 0.000,C 90.000,E1 163.142} C_DIS
LIN {X 0.098,Y -390.652,Z 693.694,A 0.000,B 0.000,C 90.000,E1 160.967} C_DIS
LIN {X -0.011,Y -390.721,Z 693.683,A 0.000,B 0.000,C 90.000,E1 158.847} C_DIS
LIN {X 0.077,Y -390.803,Z 693.675,A 0.000,B 0.000,C 90.000,E1 157.411} C_DIS
LIN {X 0.015,Y -390.939,Z 693.667,A 0.000,B 0.000,C 90.000,E1 155.997} C_DIS
LIN {X -0.216,Y -391.180,Z 693.655,A 0.000,B 0.000,C 90.000,E1 153.896} C_DIS
LIN {X -0.065,Y -391.524,Z 693.641,A 0.000,B 0.000,C 90.000,E1 151.385} C_DIS
LIN {X -0.117,Y -392.012,Z 693.631,A 0.000,B 0.000,C 90.000,E1 149.616} C_DIS
LIN {X 0.241,Y -392.636,Z 693.621,A 0.000,B 0.000,C 90.000,E1 147.788} C_DIS
LIN {X 0.021,Y -394.369,Z 693.602,A 0.000,B 0.000,C 90.000,E1 144.276} C_DIS
LIN {X 0.236,Y -395.699,Z 693.592,A 0.000,B 0.000,C 90.000,E1 142.477} C_DIS
LIN {X -0.084,Y -398.190,Z 693.576,A 0.000,B 0.000,C 90.000,E1 139.703} C_DIS
LIN {X 0.217,Y -400.285,Z 693.564,A 0.000,B 0.000,C 90.000,E1 137.553} C_DIS
LIN {X -0.043,Y -401.391,Z 693.559,A 0.000,B 0.000,C 90.000,E1 136.539} C_DIS
LIN {X 0.164,Y -402.391,Z 693.555,A 0.000,B 0.000,C 90.000,E1 135.810} C_DIS
LIN {X 0.011,Y -404.285,Z 693.550,A 0.000,B 0.000,C 90.000,E1 134.960} C_DIS
LIN {X -0.189,Y -406.254,Z 693.547,A 0.000,B 0.000,C 90.000,E1 134.433} C_DIS
LIN {X 0.086,Y -409.232,Z 693.544,A 0.000,B 0.000,C 90.000,E1 133.866} C_DIS
LIN {X 0.025,Y -413.525,Z 693.541,A 0.000,B 0.000,C 90.000,E1 133.338} C_DIS
LIN {X -0.036,Y -419.627,Z 693.537,A 0.000,B 0.000,C 90.000,E1 132.732} C_DIS
LIN {X 0.139,Y -436.120,Z 693.529,A 0.000,B 0.000,C 90.000,E1 131.229} C_DIS
LIN {X 0.015,Y -456.247,Z 693.520,A 0.000,B 0.000,C 90.000,E1 129.564} C_DIS
LIN {X -0.112,Y -463.966,Z 693.516,A 0.000,B 0.000,C 90.000,E1 128.955} C_DIS
LIN {X -0.017,Y -471.361,Z 693.513,A 0.000,B 0.000,C 90.000,E1 128.302} C_DIS
LIN {X 0.043,Y -479.955,Z 693.509,A 0.000,B 0.000,C 90.000,E1 127.523} C_DIS
LIN {X 0.081,Y -486.857,Z 693.505,A 0.000,B 0.000,C 90.000,E1 126.870} C_DIS
LIN {X -0.277,Y -495.276,Z 693.500,A 0.000,B 0.000,C 90.000,E1 126.091} C_DIS
LIN {X -0.126,Y -500.698,Z 693.497,A 0.000,B 0.000,C 90.000,E1 125.518} C_DIS
LIN {X 0.007,Y -503.326,Z 693.496,A 0.000,B 0.000,C 90.000,E1 125.231} C_DIS
LIN {X -0.235,Y -508.503,Z 693.493,A 0.000,B 0.000,C 90.000,E1 124.692} C_DIS
LIN {X 0.070,Y -513.546,Z 693.489,A 0.000,B 0.000,C 90.000,E1 124.072} C_DIS
LIN {X 0.093,Y -517.272,Z 693.487,A 0.000,B 0.000,C 90.000,E1 123.627} C_DIS
LIN {X -0.288,Y -522.653,Z 693.483,A 0.000,B 0.000,C 90.000,E1 122.959} C_DIS
LIN {X 0.190,Y -526.741,Z 693.480,A 0.000,B 0.000,C 90.000,E1 122.339} C_DIS
LIN {X -0.008,Y -529.756,Z 693.477,A 0.000,B 0.000,C 90.000,E1 121.926} C_DIS
LIN {X 0.085,Y -534.896,Z 693.473,A 0.000,B 0.000,C 90.000,E1 121.052} C_DIS
LIN {X -0.352,Y -537.329,Z 693.470,A 0.000,B 0.000,C 90.000,E1 120.669} C_DIS
LIN {X -0.062,Y -541.622,Z 693.466,A 0.000,B 0.000,C 90.000,E1 119.795} C_DIS
LIN {X 0.020,Y -544.973,Z 693.462,A 0.000,B 0.000,C 90.000,E1 119.077} C_DIS
LIN {X 0.133,Y -548.118,Z 693.458,A 0.000,B 0.000,C 90.000,E1 118.359} C_DIS
LIN {X -0.080,Y -552.718,Z 693.451,A 0.000,B 0.000,C 90.000,E1 117.257} C_DIS
LIN {X -0.016,Y -555.895,Z 693.447,A 0.000,B 0.000,C 90.000,E1 116.411} C_DIS
LIN {X -0.166,Y -558.894,Z 693.442,A 0.000,B 0.000,C 90.000,E1 115.591} C_DIS
LIN {X -0.283,Y -561.655,Z 693.438,A 0.000,B 0.000,C 90.000,E1 114.771} C_DIS
LIN {X -0.051,Y -564.953,Z 693.431,A 0.000,B 0.000,C 90.000,E1 113.643} C_DIS
LIN {X -0.106,Y -567.042,Z 693.427,A 0.000,B 0.000,C 90.000,E1 112.823} C_DIS
LIN {X -0.174,Y -568.327,Z 693.424,A 0.000,B 0.000,C 90.000,E1 112.280} C_DIS
LIN {X -0.242,Y -571.088,Z 693.416,A 0.000,B 0.000,C 90.000,E1 110.918} C_DIS
LIN {X -0.094,Y -573.085,Z 693.410,A 0.000,B 0.000,C 90.000,E1 109.812} C_DIS
LIN {X 0.251,Y -575.458,Z 693.403,A 0.000,B 0.000,C 90.000,E1 108.417} C_DIS
LIN {X -0.091,Y -577.822,Z 693.395,A 0.000,B 0.000,C 90.000,E1 107.094} C_DIS
LIN {X 0.159,Y -580.080,Z 693.387,A 0.000,B 0.000,C 90.000,E1 105.717} C_DIS
LIN {X -0.082,Y -581.834,Z 693.381,A 0.000,B 0.000,C 90.000,E1 104.662} C_DIS
LIN {X -0.243,Y -584.350,Z 693.372,A 0.000,B 0.000,C 90.000,E1 103.063} C_DIS
LIN {X -0.241,Y -587.280,Z 693.362,A 0.000,B 0.000,C 90.000,E1 101.186} C_DIS
LIN {X -0.227,Y -589.417,Z 693.355,A 0.000,B 0.000,C 90.000,E1 99.849} C_DIS
LIN {X -0.177,Y -591.319,Z 693.347,A 0.000,B 0.000,C 90.000,E1 98.511} C_DIS
LIN {X -0.183,Y -593.099,Z 693.340,A 0.000,B 0.000,C 90.000,E1 97.182} C_DIS
LIN {X -0.161,Y -594.778,Z 693.332,A 0.000,B 0.000,C 90.000,E1 95.853} C_DIS
LIN {X 0.045,Y -596.704,Z 693.324,A 0.000,B 0.000,C 90.000,E1 94.245} C_DIS
LIN {X 0.062,Y -598.148,Z 693.316,A 0.000,B 0.000,C 90.000,E1 92.922} C_DIS
LIN {X -0.193,Y -599.141,Z 693.310,A 0.000,B 0.000,C 90.000,E1 91.892} C_DIS
LIN {X -0.172,Y -600.116,Z 693.303,A 0.000,B 0.000,C 90.000,E1 90.573} C_DIS
LIN {X -0.147,Y -600.835,Z 693.296,A 0.000,B 0.000,C 90.000,E1 89.255} C_DIS
LIN {X -0.097,Y -601.367,Z 693.289,A 0.000,B 0.000,C 90.000,E1 87.936} C_DIS
LIN {X -0.313,Y -601.627,Z 693.283,A 0.000,B 0.000,C 90.000,E1 86.906} C_DIS
LIN {X -0.217,Y -601.823,Z 693.275,A 0.000,B 0.000,C 90.000,E1 85.584} C_DIS
LIN {X 0.249,Y -601.835,Z 693.270,A 0.000,B 0.000,C 90.000,E1 84.489} C_DIS
LIN {X 0.122,Y -601.746,Z 693.264,A 0.000,B 0.000,C 90.000,E1 83.451} C_DIS
LIN {X 0.214,Y -601.459,Z 693.256,A 0.000,B 0.000,C 90.000,E1 82.129} C_DIS
LIN {X 0.154,Y -601.106,Z 693.251,A 0.000,B 0.000,C 90.000,E1 81.084} C_DIS
LIN {X 0.094,Y -600.457,Z 693.245,A 0.000,B 0.000,C 90.000,E1 80.038} C_DIS
LIN {X -0.253,Y -598.911,Z 693.234,A 0.000,B 0.000,C 90.000,E1 78.229} C_DIS
LIN {X 0.066,Y -597.638,Z 693.227,A 0.000,B 0.000,C 90.000,E1 76.881} C_DIS
LIN {X -0.078,Y -596.222,Z 693.220,A 0.000,B 0.000,C 90.000,E1 75.574} C_DIS
LIN {X -0.099,Y -595.067,Z 693.214,A 0.000,B 0.000,C 90.000,E1 74.519} C_DIS
LIN {X 0.143,Y -593.085,Z 693.205,A 0.000,B 0.000,C 90.000,E1 72.906} C_DIS
LIN {X -0.162,Y -591.682,Z 693.199,A 0.000,B 0.000,C 90.000,E1 71.873} C_DIS
LIN {X -0.239,Y -589.706,Z 693.192,A 0.000,B 0.000,C 90.000,E1 70.550} C_DIS
LIN {X -0.161,Y -587.540,Z 693.184,A 0.000,B 0.000,C 90.000,E1 69.209} C_DIS
LIN {X 0.089,Y -585.075,Z 693.177,A 0.000,B 0.000,C 90.000,E1 67.847} C_DIS
LIN {X 0.022,Y -583.397,Z 693.173,A 0.000,B 0.000,C 90.000,E1 67.050} C_DIS
LIN {X 0.029,Y -580.805,Z 693.167,A 0.000,B 0.000,C 90.000,E1 65.973} C_DIS
LIN {X 0.046,Y -579.512,Z 693.164,A 0.000,B 0.000,C 90.000,E1 65.433} C_DIS
LIN {X 0.144,Y -577.356,Z 693.159,A 0.000,B 0.000,C 90.000,E1 64.613} C_DIS
LIN {X -0.046,Y -575.005,Z 693.155,A 0.000,B 0.000,C 90.000,E1 63.819} C_DIS
LIN {X 0.006,Y -572.442,Z 693.150,A 0.000,B 0.000,C 90.000,E1 62.999} C_DIS
LIN {X 0.120,Y -568.807,Z 693.144,A 0.000,B 0.000,C 90.000,E1 61.897} C_DIS
LIN {X -0.132,Y -565.838,Z 693.139,A 0.000,B 0.000,C 90.000,E1 61.101} C_DIS
LIN {X 0.080,Y -562.646,Z 693.135,A 0.000,B 0.000,C 90.000,E1 60.255} C_DIS
LIN {X 0.250,Y -559.018,Z 693.130,A 0.000,B 0.000,C 90.000,E1 59.410} C_DIS
LIN {X 0.002,Y -555.658,Z 693.126,A 0.000,B 0.000,C 90.000,E1 58.742} C_DIS
LIN {X 0.018,Y -551.917,Z 693.122,A 0.000,B 0.000,C 90.000,E1 58.043} C_DIS
LIN {X 0.173,Y -547.616,Z 693.119,A 0.000,B 0.000,C 90.000,E1 57.327} C_DIS
LIN {X -0.045,Y -543.982,Z 693.115,A 0.000,B 0.000,C 90.000,E1 56.786} C_DIS
LIN {X 0.012,Y -540.021,Z 693.112,A 0.000,B 0.000,C 90.000,E1 56.215} C_DIS
LIN {X -0.256,Y -535.585,Z 693.109,A 0.000,B 0.000,C 90.000,E1 55.674} C_DIS
LIN {X 0.056,Y -529.628,Z 693.106,A 0.000,B 0.000,C 90.000,E1 54.975} C_DIS
LIN {X 0.135,Y -525.717,Z 693.103,A 0.000,B 0.000,C 90.000,E1 54.562} C_DIS
LIN {X 0.049,Y -521.667,Z 693.101,A 0.000,B 0.000,C 90.000,E1 54.196} C_DIS
LIN {X 0.300,Y -516.226,Z 693.099,A 0.000,B 0.000,C 90.000,E1 53.703} C_DIS
LIN {X 0.243,Y -511.263,Z 693.096,A 0.000,B 0.000,C 90.000,E1 53.336} C_DIS
LIN {X 0.058,Y -503.728,Z 693.094,A 0.000,B 0.000,C 90.000,E1 52.844} C_DIS
LIN {X 0.078,Y -497.178,Z 693.091,A 0.000,B 0.000,C 90.000,E1 52.431} C_DIS
LIN {X 0.300,Y -487.334,Z 693.088,A 0.000,B 0.000,C 90.000,E1 51.823} C_DIS
LIN {X 0.156,Y -474.003,Z 693.084,A 0.000,B 0.000,C 90.000,E1 51.090} C_DIS
LIN {X 0.097,Y -462.819,Z 693.080,A 0.000,B 0.000,C 90.000,E1 50.436} C_DIS
LIN {X 0.186,Y -438.355,Z 693.072,A 0.000,B 0.000,C 90.000,E1 48.933} C_DIS
LIN {X 0.072,Y -431.860,Z 693.070,A 0.000,B 0.000,C 90.000,E1 48.528} C_DIS
LIN {X 0.202,Y -424.877,Z 693.067,A 0.000,B 0.000,C 90.000,E1 48.000} C_DIS
LIN {X 0.174,Y -424.843,Z 693.067,A 0.000,B 0.000,C 90.000,E1 48.000} C_DIS
LIN {X 0.028,Y -418.678,Z 693.049,A 0.000,B 0.000,C 90.000,E1 44.838} C_DIS
LIN {X 0.096,Y -411.760,Z 693.032,A 0.000,B 0.000,C 90.000,E1 41.757} C_DIS
LIN {X 0.063,Y -411.892,Z 693.015,A 0.000,B 0.000,C 90.000,E1 38.669} C_DIS
LIN {X 0.082,Y -413.011,Z 692.996,A 0.000,B 0.000,C 90.000,E1 35.231} C_DIS
LIN {X 0.144,Y -413.970,Z 692.984,A 0.000,B 0.000,C 90.000,E1 33.166} C_DIS
LIN {X 0.005,Y -415.062,Z 692.973,A 0.000,B 0.000,C 90.000,E1 31.131} C_DIS
LIN {X 0.085,Y -416.006,Z 692.964,A 0.000,B 0.000,C 90.000,E1 29.411} C_DIS
LIN {X -0.125,Y -417.418,Z 692.950,A 0.000,B 0.000,C 90.000,E1 27.052} C_DIS
LIN {X 0.066,Y -419.086,Z 692.937,A 0.000,B 0.000,C 90.000,E1 24.643} C_DIS
LIN {X -0.144,Y -422.030,Z 692.918,A 0.000,B 0.000,C 90.000,E1 21.280} C_DIS
LIN {X -0.041,Y -423.667,Z 692.909,A 0.000,B 0.000,C 90.000,E1 19.577} C_DIS
LIN {X 0.095,Y -425.318,Z 692.899,A 0.000,B 0.000,C 90.000,E1 17.873} C_DIS
LIN {X 0.200,Y -427.357,Z 692.888,A 0.000,B 0.000,C 90.000,E1 15.843} C_DIS
LIN {X -0.073,Y -429.992,Z 692.875,A 0.000,B 0.000,C 90.000,E1 13.536} C_DIS
LIN {X 0.236,Y -431.984,Z 692.866,A 0.000,B 0.000,C 90.000,E1 11.827} C_DIS
LIN {X 0.111,Y -434.434,Z 692.855,A 0.000,B 0.000,C 90.000,E1 9.849} C_DIS
LIN {X -0.040,Y -438.273,Z 692.838,A 0.000,B 0.000,C 90.000,E1 6.891} C_DIS
LIN {X 0.068,Y -441.867,Z 692.824,A 0.000,B 0.000,C 90.000,E1 4.245} C_DIS
LIN {X -0.050,Y -446.454,Z 692.807,A 0.000,B 0.000,C 90.000,E1 1.318} C_DIS
LIN {X -0.109,Y -451.320,Z 692.792,A 0.000,B 0.000,C 90.000,E1 358.511} C_DIS
LIN {X 0.019,Y -454.986,Z 692.781,A 0.000,B 0.000,C 90.000,E1 356.560} C_DIS
LIN {X 0.054,Y -458.109,Z 692.772,A 0.000,B 0.000,C 90.000,E1 354.951} C_DIS
LIN {X -0.081,Y -461.915,Z 692.761,A 0.000,B 0.000,C 90.000,E1 353.053} C_DIS
LIN {X -0.018,Y -465.571,Z 692.751,A 0.000,B 0.000,C 90.000,E1 351.141} C_DIS
LIN {X 0.126,Y -467.942,Z 692.744,A 0.000,B 0.000,C 90.000,E1 349.859} C_DIS
LIN {X 0.129,Y -470.773,Z 692.735,A 0.000,B 0.000,C 90.000,E1 348.285} C_DIS
LIN {X -0.180,Y -473.598,Z 692.726,A 0.000,B 0.000,C 90.000,E1 346.756} C_DIS
LIN {X -0.022,Y -477.051,Z 692.716,A 0.000,B 0.000,C 90.000,E1 344.866} C_DIS
LIN {X 0.182,Y -481.239,Z 692.704,A 0.000,B 0.000,C 90.000,E1 342.670} C_DIS
LIN {X 0.006,Y -484.286,Z 692.695,A 0.000,B 0.000,C 90.000,E1 341.148} C_DIS
LIN {X -0.104,Y -487.413,Z 692.687,A 0.000,B 0.000,C 90.000,E1 339.625} C_DIS
LIN {X -0.100,Y -491.785,Z 692.675,A 0.000,B 0.000,C 90.000,E1 337.486} C_DIS
LIN {X 0.206,Y -493.739,Z 692.670,A 0.000,B 0.000,C 90.000,E1 336.538} C_DIS
LIN {X -0.113,Y -496.006,Z 692.665,A 0.000,B 0.000,C 90.000,E1 335.665} C_DIS
LIN {X 0.043,Y -498.185,Z 692.661,A 0.000,B 0.000,C 90.000,E1 335.049} C_DIS
LIN {X -0.213,Y -499.676,Z 692.660,A 0.000,B 0.000,C 90.000,E1 334.793} C_DIS
LIN {X -0.105,Y -500.920,Z 692.659,A 0.000,B 0.000,C 90.000,E1 334.588} C_DIS
LIN {X -0.043,Y -503.444,Z 692.657,A 0.000,B 0.000,C 90.000,E1 334.280} C_DIS
LIN {X -0.204,Y -504.709,Z 692.656,A 0.000,B 0.000,C 90.000,E1 334.152} C_DIS
LIN {X -0.093,Y -508.364,Z 692.655,A 0.000,B 0.000,C 90.000,E1 333.819} C_DIS
LIN {X 0.179,Y -514.291,Z 692.652,A 0.000,B 0.000,C 90.000,E1 333.332} C_DIS
LIN {X -0.295,Y -531.358,Z 692.646,A 0.000,B 0.000,C 90.000,E1 332.231} C_DIS
LIN {X 0.090,Y -537.519,Z 692.643,A 0.000,B 0.000,C 90.000,E1 331.769} C_DIS
LIN {X -0.312,Y -544.790,Z 692.640,A 0.000,B 0.000,C 90.000,E1 331.257} C_DIS
LIN {X -0.234,Y -550.423,Z 692.638,A 0.000,B 0.000,C 90.000,E1 330.795} C_DIS
LIN {X 0.032,Y -555.939,Z 692.635,A 0.000,B 0.000,C 90.000,E1 330.284} C_DIS
LIN {X -0.068,Y -564.013,Z 692.631,A 0.000,B 0.000,C 90.000,E1 329.537} C_DIS
LIN {X 0.022,Y -573.042,Z 692.626,A 0.000,B 0.000,C 90.000,E1 328.614} C_DIS
LIN {X 0.269,Y -581.821,Z 692.621,A 0.000,B 0.000,C 90.000,E1 327.661} C_DIS
LIN {X -0.293,Y -589.187,Z 692.616,A 0.000,B 0.000,C 90.000,E1 326.914} C_DIS
LIN {X -0.015,Y -596.298,Z 692.612,A 0.000,B 0.000,C 90.000,E1 326.087} C_DIS
LIN {X -0.151,Y -603.213,Z 692.607,A 0.000,B 0.000,C 90.000,E1 325.308} C_DIS
LIN {X 0.282,Y -609.508,Z 692.603,A 0.000,B 0.000,C 90.000,E1 324.482} C_DIS
LIN {X -0.009,Y -613.430,Z 692.600,A 0.000,B 0.000,C 90.000,E1 323.989} C_DIS
LIN {X 0.000,Y -619.979,Z 692.595,A 0.000,B 0.000,C 90.000,E1 323.084} C_DIS
LIN {X 0.148,Y -623.532,Z 692.592,A 0.000,B 0.000,C 90.000,E1 322.557} C_DIS
LIN {X 0.124,Y -630.929,Z 692.586,A 0.000,B 0.000,C 90.000,E1 321.412} C_DIS
LIN {X -0.149,Y -634.845,Z 692.582,A 0.000,B 0.000,C 90.000,E1 320.803} C_DIS
LIN {X -0.001,Y -639.985,Z 692.577,A 0.000,B 0.000,C 90.000,E1 319.908} C_DIS
LIN {X 0.131,Y -646.359,Z 692.571,A 0.000,B 0.000,C 90.000,E1 318.771} C_DIS
LIN {X -0.013,Y -649.677,Z 692.568,A 0.000,B 0.000,C 90.000,E1 318.162} C_DIS
LIN {X 0.306,Y -653.649,Z 692.563,A 0.000,B 0.000,C 90.000,E1 317.391} C_DIS
LIN {X -0.264,Y -657.324,Z 692.559,A 0.000,B 0.000,C 90.000,E1 316.701} C_DIS
LIN {X -0.356,Y -660.788,Z 692.555,A 0.000,B 0.000,C 90.000,E1 315.972} C_DIS
LIN {X 0.058,Y -663.990,Z 692.551,A 0.000,B 0.000,C 90.000,E1 315.202} C_DIS
LIN {X 0.027,Y -668.001,Z 692.546,A 0.000,B 0.000,C 90.000,E1 314.231} C_DIS
LIN {X 0.072,Y -671.813,Z 692.540,A 0.000,B 0.000,C 90.000,E1 313.257} C_DIS
LIN {X 0.143,Y -675.594,Z 692.535,A 0.000,B 0.000,C 90.000,E1 312.285} C_DIS
LIN {X 0.307,Y -679.183,Z 692.530,A 0.000,B 0.000,C 90.000,E1 311.310} C_DIS
LIN {X -0.071,Y -680.945,Z 692.527,A 0.000,B 0.000,C 90.000,E1 310.862} C_DIS
LIN {X 0.170,Y -684.025,Z 692.522,A 0.000,B 0.000,C 90.000,E1 309.886} C_DIS
LIN {X -0.083,Y -686.943,Z 692.516,A 0.000,B 0.000,C 90.000,E1 308.955} C_DIS
LIN {X -0.206,Y -689.360,Z 692.511,A 0.000,B 0.000,C 90.000,E1 308.016} C_DIS
LIN {X 0.070,Y -691.034,Z 692.507,A 0.000,B 0.000,C 90.000,E1 307.282} C_DIS
LIN {X -0.054,Y -692.531,Z 692.503,A 0.000,B 0.000,C 90.000,E1 306.583} C_DIS
LIN {X -0.108,Y -694.444,Z 692.498,A 0.000,B 0.000,C 90.000,E1 305.644} C_DIS
LIN {X 0.025,Y -696.087,Z 692.493,A 0.000,B 0.000,C 90.000,E1 304.692} C_DIS
LIN {X 0.236,Y -697.781,Z 692.486,A 0.000,B 0.000,C 90.000,E1 303.499} C_DIS
LIN {X 0.422,Y -698.870,Z 692.481,A 0.000,B 0.000,C 90.000,E1 302.546} C_DIS
LIN {X 0.204,Y -700.527,Z 692.472,A 0.000,B 0.000,C 90.000,E1 300.924} C_DIS
LIN {X -0.209,Y -701.067,Z 692.468,A 0.000,B 0.000,C 90.000,E1 300.256} C_DIS
LIN {X 0.201,Y -701.800,Z 692.460,A 0.000,B 0.000,C 90.000,E1 298.821} C_DIS
LIN {X -0.040,Y -702.583,Z 692.451,A 0.000,B 0.000,C 90.000,E1 297.206} C_DIS
LIN {X 0.083,Y -703.468,Z 692.443,A 0.000,B 0.000,C 90.000,E1 295.796} C_DIS
LIN {X 0.015,Y -703.524,Z 692.441,A 0.000,B 0.000,C 90.000,E1 295.335} C_DIS
LIN {X 0.297,Y -703.444,Z 692.440,A 0.000,B 0.000,C 90.000,E1 295.079} C_DIS
LIN {X -0.355,Y -703.030,Z 692.438,A 0.000,B 0.000,C 90.000,E1 294.899} C_DIS
LIN {X 0.206,Y -701.811,Z 692.436,A 0.000,B 0.000,C 90.000,E1 294.387} C_DIS
LIN {X 0.056,Y -701.249,Z 692.435,A 0.000,B 0.000,C 90.000,E1 294.283} C_DIS
LIN {X -0.171,Y -698.505,Z 692.433,A 0.000,B 0.000,C 90.000,E1 293.951} C_DIS
LIN {X 0.093,Y -696.363,Z 692.432,A 0.000,B 0.000,C 90.000,E1 293.695} C_DIS
LIN {X -0.057,Y -694.829,Z 692.431,A 0.000,B 0.000,C 90.000,E1 293.590} C_DIS
LIN {X 0.062,Y -690.618,Z 692.430,A 0.000,B 0.000,C 90.000,E1 293.387} C_DIS
LIN {X -0.221,Y -688.766,Z 692.430,A 0.000,B 0.000,C 90.000,E1 293.334} C_DIS
LIN {X -0.316,Y -684.293,Z 692.429,A 0.000,B 0.000,C 90.000,E1 293.206} C_DIS
LIN {X 0.020,Y -679.379,Z 692.428,A 0.000,B 0.000,C 90.000,E1 293.078} C_DIS
LIN {X -0.132,Y -668.265,Z 692.427,A 0.000,B 0.000,C 90.000,E1 292.950} C_DIS
LIN {X 0.063,Y -659.717,Z 692.427,A 0.000,B 0.000,C 90.000,E1 292.823} C_DIS
LIN {X 0.263,Y -646.065,Z 692.426,A 0.000,B 0.000,C 90.000,E1 292.589} C_DIS
LIN {X 0.107,Y -636.114,Z 692.425,A 0.000,B 0.000,C 90.000,E1 292.408} C_DIS
LIN {X 0.074,Y -622.787,Z 692.423,A 0.000,B 0.000,C 90.000,E1 292.099} C_DIS
LIN {X -0.192,Y -605.780,Z 692.420,A 0.000,B 0.000,C 90.000,E1 291.663} C_DIS
LIN {X 0.064,Y -576.250,Z 692.415,A 0.000,B 0.000,C 90.000,E1 290.737} C_DIS
LIN {X 0.174,Y -564.212,Z 692.413,A 0.000,B 0.000,C 90.000,E1 290.375} C_DIS
LIN {X -0.156,Y -561.296,Z 692.413,A 0.000,B 0.000,C 90.000,E1 290.301} C_DIS
LIN {X 0.098,Y -557.987,Z 692.412,A 0.000,B 0.000,C 90.000,E1 290.120} C_DIS
LIN {X 0.155,Y -555.502,Z 692.411,A 0.000,B 0.000,C 90.000,E1 289.885} C_DIS
LIN {X 0.115,Y -555.485,Z 692.411,A 0.000,B 0.000,C 90.000,E1 289.885} C_DIS
LIN {X -0.081,Y -554.829,Z 692.409,A 0.000,B 0.000,C 90.000,E1 289.685} C_DIS
LIN {X 0.180,Y -554.351,Z 692.407,A 0.000,B 0.000,C 90.000,E1 289.214} C_DIS
LIN {X 0.181,Y -553.909,Z 692.399,A 0.000,B 0.000,C 90.000,E1 287.819} C_DIS
LIN {X 0.117,Y -553.287,Z 692.390,A 0.000,B 0.000,C 90.000,E1 286.150} C_DIS
LIN {X -0.190,Y -552.924,Z 692.384,A 0.000,B 0.000,C 90.000,E1 285.064} C_DIS
LIN {X -0.006,Y -552.396,Z 692.376,A 0.000,B 0.000,C 90.000,E1 283.647} C_DIS
LIN {X 0.164,Y -551.655,Z 692.367,A 0.000,B 0.000,C 90.000,E1 281.951} C_DIS
LIN {X -0.107,Y -550.730,Z 692.356,A 0.000,B 0.000,C 90.000,E1 280.018} C_DIS
LIN {X 0.053,Y -549.850,Z 692.343,A 0.000,B 0.000,C 90.000,E1 277.757} C_DIS
LIN {X 0.056,Y -549.274,Z 692.331,A 0.000,B 0.000,C 90.000,E1 275.511} C_DIS
LIN {X -0.044,Y -549.055,Z 692.320,A 0.000,B 0.000,C 90.000,E1 273.555} C_DIS
LIN {X 0.181,Y -548.889,Z 692.314,A 0.000,B 0.000,C 90.000,E1 272.407} C_DIS
LIN {X -0.099,Y -548.428,Z 692.306,A 0.000,B 0.000,C 90.000,E1 271.031} C_DIS
LIN {X 0.149,Y -547.661,Z 692.298,A 0.000,B 0.000,C 90.000,E1 269.599} C_DIS
LIN {X -0.107,Y -546.692,Z 692.289,A 0.000,B 0.000,C 90.000,E1 267.936} C_DIS
LIN {X 0.159,Y -545.617,Z 692.279,A 0.000,B 0.000,C 90.000,E1 266.216} C_DIS
LIN {X -0.146,Y -544.583,Z 692.271,A 0.000,B 0.000,C 90.000,E1 264.837} C_DIS
LIN {X 0.143,Y -543.250,Z 692.262,A 0.000,B 0.000,C 90.000,E1 263.109} C_DIS
LIN {X 0.002,Y -541.221,Z 692.251,A 0.000,B 0.000,C 90.000,E1 261.141} C_DIS
LIN {X 0.115,Y -538.633,Z 692.235,A 0.000,B 0.000,C 90.000,E1 258.285} C_DIS
LIN {X 0.043,Y -536.883,Z 692.224,A 0.000,B 0.000,C 90.000,E1 256.297} C_DIS
LIN {X -0.119,Y -535.885,Z 692.218,A 0.000,B 0.000,C 90.000,E1 255.172} C_DIS
LIN {X -0.150,Y -534.772,Z 692.211,A 0.000,B 0.000,C 90.000,E1 254.031} C_DIS
LIN {X -0.115,Y -532.985,Z 692.202,A 0.000,B 0.000,C 90.000,E1 252.308} C_DIS
LIN {X 0.196,Y -531.235,Z 692.192,A 0.000,B 0.000,C 90.000,E1 250.550} C_DIS
LIN {X 0.087,Y -530.292,Z 692.187,A 0.000,B 0.000,C 90.000,E1 249.699} C_DIS
LIN {X 0.150,Y -528.724,Z 692.181,A 0.000,B 0.000,C 90.000,E1 248.539} C_DIS
LIN {X 0.074,Y -526.707,Z 692.173,A 0.000,B 0.000,C 90.000,E1 247.102} C_DIS
LIN {X 0.281,Y -524.961,Z 692.166,A 0.000,B 0.000,C 90.000,E1 245.921} C_DIS
LIN {X 0.039,Y -522.055,Z 692.157,A 0.000,B 0.000,C 90.000,E1 244.204} C_DIS
LIN {X -0.076,Y -519.868,Z 692.150,A 0.000,B 0.000,C 90.000,E1 243.050} C_DIS
LIN {X -0.191,Y -516.438,Z 692.141,A 0.000,B 0.000,C 90.000,E1 241.307} C_DIS
LIN {X -0.058,Y -514.678,Z 692.136,A 0.000,B 0.000,C 90.000,E1 240.411} C_DIS
LIN {X -0.240,Y -510.916,Z 692.126,A 0.000,B 0.000,C 90.000,E1 238.663} C_DIS
LIN {X -0.024,Y -508.352,Z 692.119,A 0.000,B 0.000,C 90.000,E1 237.454} C_DIS
LIN {X -0.277,Y -505.714,Z 692.113,A 0.000,B 0.000,C 90.000,E1 236.294} C_DIS
LIN {X 0.015,Y -502.319,Z 692.104,A 0.000,B 0.000,C 90.000,E1 234.769} C_DIS
LIN {X -0.047,Y -499.524,Z 692.098,A 0.000,B 0.000,C 90.000,E1 233.577} C_DIS
LIN {X 0.144,Y -496.574,Z 692.091,A 0.000,B 0.000,C 90.000,E1 232.351} C_DIS
LIN {X 0.310,Y -490.600,Z 692.078,A 0.000,B 0.000,C 90.000,E1 229.908} C_DIS
LIN {X 0.099,Y -485.513,Z 692.066,A 0.000,B 0.000,C 90.000,E1 227.796} C_DIS
LIN {X -0.079,Y -481.286,Z 692.055,A 0.000,B 0.000,C 90.000,E1 225.972} C_DIS
LIN {X -0.248,Y -478.560,Z 692.049,A 0.000,B 0.000,C 90.000,E1 224.757} C_DIS
LIN {X 0.100,Y -474.232,Z 692.038,A 0.000,B 0.000,C 90.000,E1 222.852} C_DIS
LIN {X 0.020,Y -470.077,Z 692.028,A 0.000,B 0.000,C 90.000,E1 220.987} C_DIS
LIN {X 0.063,Y -467.395,Z 692.021,A 0.000,B 0.000,C 90.000,E1 219.725} C_DIS
LIN {X 0.233,Y -463.390,Z 692.010,A 0.000,B 0.000,C 90.000,E1 217.810} C_DIS
LIN {X -0.018,Y -457.110,Z 691.993,A 0.000,B 0.000,C 90.000,E1 214.659} C_DIS
LIN {X 0.026,Y -454.640,Z 691.985,A 0.000,B 0.000,C 90.000,E1 213.372} C_DIS
LIN {X 0.136,Y -451.590,Z 691.977,A 0.000,B 0.000,C 90.000,E1 211.750} C_DIS
LIN {X 0.114,Y -447.302,Z 691.964,A 0.000,B 0.000,C 90.000,E1 209.489} C_DIS
LIN {X 0.146,Y -443.215,Z 691.951,A 0.000,B 0.000,C 90.000,E1 207.206} C_DIS
LIN {X -0.024,Y -440.218,Z 691.942,A 0.000,B 0.000,C 90.000,E1 205.591} C_DIS
LIN {X -0.050,Y -437.254,Z 691.933,A 0.000,B 0.000,C 90.000,E1 203.951} C_DIS
LIN {X 0.092,Y -434.199,Z 691.924,A 0.000,B 0.000,C 90.000,E1 202.280} C_DIS
LIN {X 0.175,Y -431.203,Z 691.915,A 0.000,B 0.000,C 90.000,E1 200.610} C_DIS
LIN {X 0.245,Y -427.519,Z 691.904,A 0.000,B 0.000,C 90.000,E1 198.598} C_DIS
LIN {X -0.074,Y -422.753,Z 691.889,A 0.000,B 0.000,C 90.000,E1 195.953} C_DIS
LIN {X 0.062,Y -419.807,Z 691.879,A 0.000,B 0.000,C 90.000,E1 194.245} C_DIS
LIN {X -0.205,Y -416.223,Z 691.868,A 0.000,B 0.000,C 90.000,E1 192.243} C_DIS
LIN {X 0.126,Y -413.432,Z 691.858,A 0.000,B 0.000,C 90.000,E1 190.489} C_DIS
LIN {X -0.020,Y -409.605,Z 691.845,A 0.000,B 0.000,C 90.000,E1 188.106} C_DIS
LIN {X 0.005,Y -406.503,Z 691.834,A 0.000,B 0.000,C 90.000,E1 186.030} C_DIS
LIN {X -0.048,Y -403.563,Z 691.822,A 0.000,B 0.000,C 90.000,E1 183.955} C_DIS
LIN {X 0.072,Y -400.086,Z 691.806,A 0.000,B 0.000,C 90.000,E1 181.146} C_DIS
LIN {X 0.023,Y -396.872,Z 691.789,A 0.000,B 0.000,C 90.000,E1 177.993} C_DIS
LIN {X 0.015,Y -394.897,Z 691.775,A 0.000,B 0.000,C 90.000,E1 175.527} C_DIS
LIN {X 0.143,Y -392.526,Z 691.750,A 0.000,B 0.000,C 90.000,E1 170.905} C_DIS
LIN {X -0.164,Y -391.902,Z 691.736,A 0.000,B 0.000,C 90.000,E1 168.465} C_DIS
LIN {X 0.142,Y -391.510,Z 691.726,A 0.000,B 0.000,C 90.000,E1 166.645} C_DIS
LIN {X 0.155,Y -390.928,Z 691.706,A 0.000,B 0.000,C 90.000,E1 163.087} C_DIS
LIN {X 0.099,Y -390.933,Z 691.692,A 0.000,B 0.000,C 90.000,E1 160.604} C_DIS
LIN {X -0.147,Y -391.084,Z 691.677,A 0.000,B 0.000,C 90.000,E1 157.794} C_DIS
LIN {X -0.179,Y -391.225,Z 691.665,A 0.000,B 0.000,C 90.000,E1 155.665} C_DIS
LIN {X 0.153,Y -391.490,Z 691.651,A 0.000,B 0.000,C 90.000,E1 153.127} C_DIS
LIN {X 0.016,Y -392.187,Z 691.633,A 0.000,B 0.000,C 90.000,E1 149.950} C_DIS
LIN {X 0.234,Y -392.878,Z 691.621,A 0.000,B 0.000,C 90.000,E1 147.788} C_DIS
LIN {X -0.034,Y -395.096,Z 691.598,A 0.000,B 0.000,C 90.000,E1 143.577} C_DIS
LIN {X 0.180,Y -397.333,Z 691.582,A 0.000,B 0.000,C 90.000,E1 140.723} C_DIS
LIN {X 0.013,Y -399.644,Z 691.568,A 0.000,B 0.000,C 90.000,E1 138.286} C_DIS
LIN {X -0.030,Y -401.361,Z 691.559,A 0.000,B 0.000,C 90.000,E1 136.539} C_DIS
LIN {X 0.177,Y -402.252,Z 691.555,A 0.000,B 0.000,C 90.000,E1 135.810} C_DIS
LIN {X -0.192,Y -403.964,Z 691.550,A 0.000,B 0.000,C 90.000,E1 135.000} C_DIS
LIN {X -0.118,Y -406.223,Z 691.546,A 0.000,B 0.000,C 90.000,E1 134.271} C_DIS
LIN {X 0.222,Y -409.037,Z 691.543,A 0.000,B 0.000,C 90.000,E1 133.704} C_DIS
LIN {X 0.067,Y -411.591,Z 691.541,A 0.000,B 0.000,C 90.000,E1 133.380} C_DIS
LIN {X -0.083,Y -414.682,Z 691.539,A 0.000,B 0.000,C 90.000,E1 133.056} C_DIS
LIN {X 0.077,Y -421.969,Z 691.535,A 0.000,B 0.000,C 90.000,E1 132.324} C_DIS
LIN {X 0.041,Y -444.963,Z 691.524,A 0.000,B 0.000,C 90.000,E1 130.334} C_DIS
LIN {X 0.018,Y -463.511,Z 691.516,A 0.000,B 0.000,C 90.000,E1 128.830} C_DIS
LIN {X -0.086,Y -469.434,Z 691.513,A 0.000,B 0.000,C 90.000,E1 128.338} C_DIS
LIN {X -0.280,Y -479.760,Z 691.508,A 0.000,B 0.000,C 90.000,E1 127.443} C_DIS
LIN {X -0.030,Y -486.893,Z 691.504,A 0.000,B 0.000,C 90.000,E1 126.744} C_DIS
LIN {X -0.262,Y -493.951,Z 691.500,A 0.000,B 0.000,C 90.000,E1 126.091} C_DIS
LIN {X -0.073,Y -499.423,Z 691.497,A 0.000,B 0.000,C 90.000,E1 125.518} C_DIS
LIN {X -0.120,Y -506.135,Z 691.493,A 0.000,B 0.000,C 90.000,E1 124.818} C_DIS
LIN {X 0.059,Y -512.605,Z 691.489,A 0.000,B 0.000,C 90.000,E1 124.072} C_DIS
LIN {X 0.097,Y -516.374,Z 691.487,A 0.000,B 0.000,C 90.000,E1 123.627} C_DIS
LIN {X 0.104,Y -521.012,Z 691.484,A 0.000,B 0.000,C 90.000,E1 123.038} C_DIS
LIN {X -0.007,Y -525.371,Z 691.480,A 0.000,B 0.000,C 90.000,E1 122.467} C_DIS
LIN {X 0.073,Y -529.422,Z 691.477,A 0.000,B 0.000,C 90.000,E1 121.878} C_DIS
LIN {X -0.140,Y -533.911,Z 691.473,A 0.000,B 0.000,C 90.000,E1 121.180} C_DIS
LIN {X 0.017,Y -537.905,Z 691.469,A 0.000,B 0.000,C 90.000,E1 120.463} C_DIS
LIN {X 0.063,Y -541.562,Z 691.465,A 0.000,B 0.000,C 90.000,E1 119.745} C_DIS
LIN {X 0.147,Y -544.968,Z 691.461,A 0.000,B 0.000,C 90.000,E1 119.027} C_DIS
LIN {X 0.144,Y -548.732,Z 691.457,A 0.000,B 0.000,C 90.000,E1 118.180} C_DIS
LIN {X -0.078,Y -551.163,Z 691.454,A 0.000,B 0.000,C 90.000,E1 117.641} C_DIS
LIN {X -0.030,Y -554.478,Z 691.449,A 0.000,B 0.000,C 90.000,E1 116.796} C_DIS
LIN {X 0.093,Y -558.561,Z 691.443,A 0.000,B 0.000,C 90.000,E1 115.668} C_DIS
LIN {X -0.022,Y -561.395,Z 691.438,A 0.000,B 0.000,C 90.000,E1 114.847} C_DIS
LIN {X -0.303,Y -564.765,Z 691.432,A 0.000,B 0.000,C 90.000,E1 113.770} C_DIS
LIN {X -0.170,Y -566.318,Z 691.429,A 0.000,B 0.000,C 90.000,E1 113.206} C_DIS
LIN {X -0.213,Y -568.306,Z 691.424,A 0.000,B 0.000,C 90.000,E1 112.386} C_DIS
LIN {X 0.242,Y -571.127,Z 691.417,A 0.000,B 0.000,C 90.000,E1 110.972} C_DIS
LIN {X 0.193,Y -573.163,Z 691.411,A 0.000,B 0.000,C 90.000,E1 109.885} C_DIS
LIN {X 0.003,Y -575.563,Z 691.403,A 0.000,B 0.000,C 90.000,E1 108.544} C_DIS
LIN {X -0.332,Y -577.959,Z 691.396,A 0.000,B 0.000,C 90.000,E1 107.221} C_DIS
LIN {X 0.142,Y -580.712,Z 691.387,A 0.000,B 0.000,C 90.000,E1 105.552} C_DIS
LIN {X 0.064,Y -582.464,Z 691.381,A 0.000,B 0.000,C 90.000,E1 104.481} C_DIS
LIN {X 0.243,Y -584.577,Z 691.373,A 0.000,B 0.000,C 90.000,E1 103.119} C_DIS
LIN {X -0.075,Y -588.035,Z 691.361,A 0.000,B 0.000,C 90.000,E1 101.007} C_DIS
LIN {X 0.207,Y -590.522,Z 691.352,A 0.000,B 0.000,C 90.000,E1 99.378} C_DIS
LIN {X 0.184,Y -592.420,Z 691.345,A 0.000,B 0.000,C 90.000,E1 98.049} C_DIS
LIN {X 0.199,Y -594.205,Z 691.337,A 0.000,B 0.000,C 90.000,E1 96.720} C_DIS
LIN {X 0.237,Y -595.861,Z 691.330,A 0.000,B 0.000,C 90.000,E1 95.391} C_DIS
LIN {X 0.196,Y -597.468,Z 691.323,A 0.000,B 0.000,C 90.000,E1 94.073} C_DIS
LIN {X 0.228,Y -598.904,Z 691.315,A 0.000,B 0.000,C 90.000,E1 92.751} C_DIS
LIN {X 0.004,Y -599.852,Z 691.310,A 0.000,B 0.000,C 90.000,E1 91.718} C_DIS
LIN {X 0.020,Y -600.821,Z 691.302,A 0.000,B 0.000,C 90.000,E1 90.401} C_DIS
LIN {X -0.192,Y -601.394,Z 691.296,A 0.000,B 0.000,C 90.000,E1 89.370} C_DIS
LIN {X -0.132,Y -601.953,Z 691.289,A 0.000,B 0.000,C 90.000,E1 88.051} C_DIS
LIN {X 0.262,Y -602.244,Z 691.283,A 0.000,B 0.000,C 90.000,E1 86.963} C_DIS
LIN {X 0.014,Y -602.459,Z 691.275,A 0.000,B 0.000,C 90.000,E1 85.412} C_DIS
LIN {X -0.113,Y -602.425,Z 691.269,A 0.000,B 0.000,C 90.000,E1 84.375} C_DIS
LIN {X -0.235,Y -602.289,Z 691.263,A 0.000,B 0.000,C 90.000,E1 83.337} C_DIS
LIN {X 0.236,Y -602.054,Z 691.257,A 0.000,B 0.000,C 90.000,E1 82.243} C_DIS
LIN {X 0.187,Y -601.720,Z 691.251,A 0.000,B 0.000,C 90.000,E1 81.197} C_DIS
LIN {X 0.137,Y -601.041,Z 691.245,A 0.000,B 0.000,C 90.000,E1 80.151} C_DIS
LIN {X -0.208,Y -599.917,Z 691.238,A 0.000,B 0.000,C 90.000,E1 78.870} C_DIS
LIN {X -0.168,Y -598.979,Z 691.232,A 0.000,B 0.000,C 90.000,E1 77.813} C_DIS
LIN {X 0.156,Y -597.630,Z 691.225,A 0.000,B 0.000,C 90.000,E1 76.464} C_DIS
LIN {X -0.135,Y -596.185,Z 691.218,A 0.000,B 0.000,C 90.000,E1 75.172} C_DIS
LIN {X -0.007,Y -594.906,Z 691.212,A 0.000,B 0.000,C 90.000,E1 74.102} C_DIS
LIN {X 0.099,Y -593.595,Z 691.206,A 0.000,B 0.000,C 90.000,E1 73.032} C_DIS
LIN {X 0.047,Y -591.773,Z 691.198,A 0.000,B 0.000,C 90.000,E1 71.710} C_DIS
LIN {X 0.155,Y -589.744,Z 691.191,A 0.000,B 0.000,C 90.000,E1 70.369} C_DIS
LIN {X -0.193,Y -587.937,Z 691.185,A 0.000,B 0.000,C 90.000,E1 69.337} C_DIS
LIN {X 0.061,Y -585.463,Z 691.178,A 0.000,B 0.000,C 90.000,E1 67.975} C_DIS
LIN {X -0.004,Y -583.769,Z 691.173,A 0.000,B 0.000,C 90.000,E1 67.177} C_DIS
LIN {X 0.008,Y -581.198,Z 691.167,A 0.000,B 0.000,C 90.000,E1 66.102} C_DIS
LIN {X 0.131,Y -579.125,Z 691.163,A 0.000,B 0.000,C 90.000,E1 65.281} C_DIS
LIN {X 0.232,Y -576.892,Z 691.158,A 0.000,B 0.000,C 90.000,E1 64.460} C_DIS
LIN {X 0.306,Y -574.456,Z 691.154,A 0.000,B 0.000,C 90.000,E1 63.640} C_DIS
LIN {X -0.323,Y -570.919,Z 691.148,A 0.000,B 0.000,C 90.000,E1 62.615} C_DIS
LIN {X -0.056,Y -568.059,Z 691.143,A 0.000,B 0.000,C 90.000,E1 61.769} C_DIS
LIN {X 0.179,Y -565.004,Z 691.139,A 0.000,B 0.000,C 90.000,E1 60.923} C_DIS
LIN {X 0.081,Y -562.820,Z 691.136,A 0.000,B 0.000,C 90.000,E1 60.383} C_DIS
LIN {X 0.151,Y -558.541,Z 691.130,A 0.000,B 0.000,C 90.000,E1 59.410} C_DIS
LIN {X -0.101,Y -555.055,Z 691.126,A 0.000,B 0.000,C 90.000,E1 58.742} C_DIS
LIN {X -0.017,Y -551.220,Z 691.122,A 0.000,B 0.000,C 90.000,E1 58.043} C_DIS
LIN {X 0.258,Y -547.783,Z 691.119,A 0.000,B 0.000,C 90.000,E1 57.454} C_DIS
LIN {X 0.043,Y -544.105,Z 691.116,A 0.000,B 0.000,C 90.000,E1 56.914} C_DIS
LIN {X 0.101,Y -540.085,Z 691.113,A 0.000,B 0.000,C 90.000,E1 56.342} C_DIS
LIN {X -0.166,Y -535.622,Z 691.110,A 0.000,B 0.000,C 90.000,E1 55.801} C_DIS
LIN {X 0.285,Y -530.585,Z 691.107,A 0.000,B 0.000,C 90.000,E1 55.182} C_DIS
LIN {X -0.249,Y -525.143,Z 691.104,A 0.000,B 0.000,C 90.000,E1 54.689} C_DIS
LIN {X -0.044,Y -520.815,Z 691.102,A 0.000,B 0.000,C 90.000,E1 54.276} C_DIS
LIN {X -0.076,Y -514.740,Z 691.099,A 0.000,B 0.000,C 90.000,E1 53.783} C_DIS
LIN {X 0.045,Y -509.922,Z 691.097,A 0.000,B 0.000,C 90.000,E1 53.417} C_DIS
LIN {X 0.001,Y -501.753,Z 691.094,A 0.000,B 0.000,C 90.000,E1 52.889} C_DIS
LIN {X 0.277,Y -496.902,Z 691.092,A 0.000,B 0.000,C 90.000,E1 52.557} C_DIS
LIN {X -0.076,Y -488.565,Z 691.089,A 0.000,B 0.000,C 90.000,E1 52.110} C_DIS
LIN {X 0.094,Y -468.780,Z 691.083,A 0.000,B 0.000,C 90.000,E1 50.964} C_DIS
LIN {X 0.044,Y -452.243,Z 691.078,A 0.000,B 0.000,C 90.000,E1 49.989} C_DIS
LIN {X 0.033,Y -440.907,Z 691.074,A 0.000,B 0.000,C 90.000,E1 49.299} C_DIS
LIN {X -0.071,Y -429.562,Z 691.070,A 0.000,B 0.000,C 90.000,E1 48.566} C_DIS
LIN {X 0.028,Y -425.340,Z 691.068,A 0.000,B 0.000,C 90.000,E1 48.243} C_DIS
LIN {X 0.001,Y -425.324,Z 691.068,A 0.000,B 0.000,C 90.000,E1 48.243} C_DIS
LIN {X -0.095,Y -418.464,Z 691.049,A 0.000,B 0.000,C 90.000,E1 44.757} C_DIS
LIN {X 0.106,Y -412.260,Z 691.033,A 0.000,B 0.000,C 90.000,E1 42.000} C_DIS
LIN {X 0.132,Y -412.131,Z 691.030,A 0.000,B 0.000,C 90.000,E1 41.310} C_DIS
LIN {X 0.024,Y -412.500,Z 691.011,A 0.000,B 0.000,C 90.000,E1 37.890} C_DIS
LIN {X -0.024,Y -413.516,Z 690.995,A 0.000,B 0.000,C 90.000,E1 35.152} C_DIS
LIN {X -0.015,Y -414.679,Z 690.982,A 0.000,B 0.000,C 90.000,E1 32.752} C_DIS
LIN {X -0.086,Y -415.613,Z 690.972,A 0.000,B 0.000,C 90.000,E1 31.052} C_DIS
LIN {X -0.052,Y -416.731,Z 690.961,A 0.000,B 0.000,C 90.000,E1 28.999} C_DIS
LIN {X -0.018,Y -417.959,Z 690.950,A 0.000,B 0.000,C 90.000,E1 26.950} C_DIS
END
